LIN {X 0,Y 340.767,Z 675.84,A -85,B 0,C 180,E1 -14245.664,E2 -14245.664} C_VEL
LIN {X 0,Y 340.733,Z 675.796,A -85,B 0,C 180,E1 -14248.32,E2 -14248.32} C_VEL
LIN {X 0,Y 340.696,Z 675.835,A -85,B 0,C 180,E1 -14251.044,E2 -14251.044} C_VEL
LIN {X 0,Y 340.71,Z 675.812,A -85,B 0,C 180,E1 -14255.279,E2 -14255.279} C_VEL
LIN {X 0,Y 340.71,Z 675.84,A -85,B 0,C 180,E1 -14258.388,E2 -14258.388} C_VEL
LIN {X 0,Y 340.718,Z 675.858,A -85,B 0,C 180,E1 -14261.304,E2 -14261.304} C_VEL
LIN {X 0,Y 340.716,Z 675.858,A -85,B 0,C 180,E1 -14264.532,E2 -14264.532} C_VEL
LIN {X 0,Y 340.727,Z 675.857,A -85,B 0,C 180,E1 -14267.949,E2 -14267.949} C_VEL
LIN {X 0,Y 340.758,Z 676.06,A -85,B 0,C 180,E1 -14271.835,E2 -14271.835} C_VEL
LIN {X 0,Y 341.027,Z 677.234,A -85,B 0,C 180,E1 -14272.318,E2 -14272.318} C_VEL
LIN {X 0,Y 342.41,Z 679.667,A -85,B 0,C 180,E1 -14272.976,E2 -14272.976} C_VEL
LIN {X 0,Y 344.684,Z 681.388,A -85,B 0,C 180,E1 -14273.895,E2 -14273.895} C_VEL
LIN {X 0,Y 345.815,Z 682.281,A -85,B 0,C 180,E1 -14274.381,E2 -14274.381} C_VEL
LIN {X 0,Y 347.437,Z 685.007,A -85,B 0,C 180,E1 -14275.129,E2 -14275.129} C_VEL
LIN {X 0,Y 350.033,Z 687.231,A -85,B 0,C 180,E1 -14276.266,E2 -14276.266} C_VEL
LIN {X 0,Y 351.154,Z 688.02,A -85,B 0,C 180,E1 -14276.744,E2 -14276.744} C_VEL
LIN {X 0,Y 353.08,Z 690.98,A -85,B 0,C 180,E1 -14277.691,E2 -14277.691} C_VEL
LIN {X 0,Y 355.654,Z 693.147,A -85,B 0,C 180,E1 -14278.882,E2 -14278.882} C_VEL
LIN {X 0,Y 357.002,Z 694.101,A -85,B 0,C 180,E1 -14279.493,E2 -14279.493} C_VEL
LIN {X 0,Y 359.425,Z 697.413,A -85,B 0,C 180,E1 -14280.737,E2 -14280.737} C_VEL
LIN {X 0,Y 362.273,Z 699.528,A -85,B 0,C 180,E1 -14282.149,E2 -14282.149} C_VEL
LIN {X 0,Y 363.124,Z 700.378,A -85,B 0,C 180,E1 -14282.611,E2 -14282.611} C_VEL
LIN {X 0,Y 365.113,Z 703.18,A -85,B 0,C 180,E1 -14283.723,E2 -14283.723} C_VEL
LIN {X 0,Y 367.846,Z 705.386,A -85,B 0,C 180,E1 -14285.232,E2 -14285.232} C_VEL
LIN {X 0,Y 369.089,Z 706.243,A -85,B 0,C 180,E1 -14285.932,E2 -14285.932} C_VEL
LIN {X 0,Y 371.469,Z 709.532,A -85,B 0,C 180,E1 -14287.437,E2 -14287.437} C_VEL
LIN {X 0,Y 374.201,Z 711.633,A -85,B 0,C 180,E1 -14289.17,E2 -14289.17} C_VEL
LIN {X 0,Y 375.879,Z 712.69,A -85,B 0,C 180,E1 -14290.269,E2 -14290.269} C_VEL
LIN {X 0,Y 377.819,Z 715.534,A -85,B 0,C 180,E1 -14291.772,E2 -14291.772} C_VEL
LIN {X 0,Y 380.32,Z 717.676,A -85,B 0,C 180,E1 -14293.763,E2 -14293.763} C_VEL
LIN {X 0,Y 382.812,Z 719.086,A -85,B 0,C 180,E1 -14295.905,E2 -14295.905} C_VEL
LIN {X 0,Y 384.247,Z 721.472,A -85,B 0,C 180,E1 -14297.505,E2 -14297.505} C_VEL
LIN {X 0,Y 386.099,Z 723.313,A -85,B 0,C 180,E1 -14299.68,E2 -14299.68} C_VEL
LIN {X 0,Y 387.892,Z 724.36,A -85,B 0,C 180,E1 -14302.256,E2 -14302.256} C_VEL
LIN {X 0,Y 389.273,Z 725.077,A -85,B 0,C 180,E1 -14305.045,E2 -14305.045} C_VEL
LIN {X 0,Y 390.059,Z 725.483,A -85,B 0,C 180,E1 -14307.935,E2 -14307.935} C_VEL
LIN {X 0,Y 390.26,Z 725.548,A -85,B 0,C 180,E1 -14310,E2 -14310} C_VEL
LIN {X 0,Y 390.059,Z 725.486,A -85,B 0,C 180,E1 -14312.065,E2 -14312.065} C_VEL
LIN {X 0,Y 389.272,Z 725.078,A -85,B 0,C 180,E1 -14314.953,E2 -14314.953} C_VEL
LIN {X 0,Y 387.893,Z 724.36,A -85,B 0,C 180,E1 -14317.744,E2 -14317.744} C_VEL
LIN {X 0,Y 386.1,Z 723.319,A -85,B 0,C 180,E1 -14320.32,E2 -14320.32} C_VEL
LIN {X 0,Y 384.178,Z 721.341,A -85,B 0,C 180,E1 -14322.58,E2 -14322.58} C_VEL
LIN {X 0,Y 382.562,Z 718.807,A -85,B 0,C 180,E1 -14324.348,E2 -14324.348} C_VEL
LIN {X 0,Y 379.559,Z 717.133,A -85,B 0,C 180,E1 -14326.866,E2 -14326.866} C_VEL
LIN {X 0,Y 377.187,Z 714.751,A -85,B 0,C 180,E1 -14328.707,E2 -14328.707} C_VEL
LIN {X 0,Y 375.566,Z 712.349,A -85,B 0,C 180,E1 -14329.944,E2 -14329.944} C_VEL
LIN {X 0,Y 372.385,Z 710.399,A -85,B 0,C 180,E1 -14331.974,E2 -14331.974} C_VEL
LIN {X 0,Y 369.885,Z 707.552,A -85,B 0,C 180,E1 -14333.563,E2 -14333.563} C_VEL
LIN {X 0,Y 368.864,Z 705.955,A -85,B 0,C 180,E1 -14334.201,E2 -14334.201} C_VEL
LIN {X 0,Y 365.884,Z 703.986,A -85,B 0,C 180,E1 -14335.838,E2 -14335.838} C_VEL
LIN {X 0,Y 363.626,Z 701.259,A -85,B 0,C 180,E1 -14337.098,E2 -14337.098} C_VEL
LIN {X 0,Y 362.729,Z 699.764,A -85,B 0,C 180,E1 -14337.62,E2 -14337.62} C_VEL
LIN {X 0,Y 359.826,Z 697.815,A -85,B 0,C 180,E1 -14339.06,E2 -14339.06} C_VEL
LIN {X 0,Y 357.355,Z 694.737,A -85,B 0,C 180,E1 -14340.312,E2 -14340.312} C_VEL
LIN {X 0,Y 356.555,Z 693.62,A -85,B 0,C 180,E1 -14340.722,E2 -14340.722} C_VEL
LIN {X 0,Y 353.621,Z 691.552,A -85,B 0,C 180,E1 -14342.065,E2 -14342.065} C_VEL
LIN {X 0,Y 351.546,Z 688.772,A -85,B 0,C 180,E1 -14343.05,E2 -14343.05} C_VEL
LIN {X 0,Y 350.95,Z 687.687,A -85,B 0,C 180,E1 -14343.357,E2 -14343.357} C_VEL
LIN {X 0,Y 347.992,Z 685.635,A -85,B 0,C 180,E1 -14344.624,E2 -14344.624} C_VEL
LIN {X 0,Y 346.203,Z 683.113,A -85,B 0,C 180,E1 -14345.429,E2 -14345.429} C_VEL
LIN {X 0,Y 345.49,Z 681.814,A -85,B 0,C 180,E1 -14345.769,E2 -14345.769} C_VEL
LIN {X 0,Y 342.717,Z 679.998,A -85,B 0,C 180,E1 -14346.894,E2 -14346.894} C_VEL
LIN {X 0,Y 341.161,Z 677.596,A -85,B 0,C 180,E1 -14347.61,E2 -14347.61} C_VEL
LIN {X 0,Y 340.803,Z 676.233,A -85,B 0,C 180,E1 -14348.043,E2 -14348.043} C_VEL
LIN {X 0,Y 340.72,Z 675.904,A -85,B 0,C 180,E1 -14348.389,E2 -14348.389} C_VEL
LIN {X 0,Y 340.727,Z 675.857,A -85,B 0,C 180,E1 -14352.051,E2 -14352.051} C_VEL
LIN {X 0,Y 340.716,Z 675.858,A -85,B 0,C 180,E1 -14355.468,E2 -14355.468} C_VEL
LIN {X 0,Y 340.718,Z 675.858,A -85,B 0,C 180,E1 -14358.696,E2 -14358.696} C_VEL
LIN {X 0,Y 340.731,Z 675.833,A -85,B 0,C 180,E1 -14361.773,E2 -14361.773} C_VEL
LIN {X 0,Y 340.715,Z 675.827,A -85,B 0,C 180,E1 -14365.595,E2 -14365.595} C_VEL
LIN {X 0,Y 340.715,Z 675.816,A -85,B 0,C 180,E1 -14369.568,E2 -14369.568} C_VEL
LIN {X 0,Y 340.797,Z 675.806,A -85,B 0,C 180,E1 -14373.02,E2 -14373.02} C_VEL
LIN {X 0,Y 340.757,Z 675.844,A -85,B 0,C 180,E1 -14374.692,E2 -14374.692} C_VEL
LIN {X 0,Y 340.082,Z 675.936,A -85,B 0,C 180,E1 -14375.679,E2 -14375.679} C_VEL
LIN {X 0,Y 337.203,Z 676.292,A -85,B 0,C 180,E1 -14377.284,E2 -14377.284} C_VEL
LIN {X 0,Y 334.787,Z 676.588,A -85,B 0,C 180,E1 -14378.584,E2 -14378.584} C_VEL
LIN {X 0,Y 333.782,Z 676.719,A -85,B 0,C 180,E1 -14379.591,E2 -14379.591} C_VEL
LIN {X 0,Y 333.717,Z 676.723,A -85,B 0,C 180,E1 -14379.931,E2 -14379.931} C_VEL
LIN {X 0,Y 333.737,Z 676.708,A -85,B 0,C 180,E1 -14382.854,E2 -14382.854} C_VEL
LIN {X 0,Y 333.788,Z 676.698,A -85,B 0,C 180,E1 -14386.609,E2 -14386.609} C_VEL
LIN {X 0,Y 333.853,Z 676.706,A -85,B 0,C 180,E1 -14390.305,E2 -14390.305} C_VEL
LIN {X 0,Y 334.006,Z 676.673,A -85,B 0,C 180,E1 -14392.747,E2 -14392.747} C_VEL
LIN {X 0,Y 333.807,Z 676.714,A -85,B 0,C 180,E1 -14395.169,E2 -14395.169} C_VEL
LIN {X 0,Y 334.099,Z 676.658,A -85,B 0,C 180,E1 -14397.589,E2 -14397.589} C_VEL
LIN {X 0,Y 334.259,Z 676.66,A -85,B 0,C 180,E1 -14400,E2 -14400} C_VEL
LIN {X 0,Y 334.099,Z 676.662,A -85,B 0,C 180,E1 -14402.412,E2 -14402.412} C_VEL
LIN {X 0,Y 334.012,Z 676.688,A -85,B 0,C 180,E1 -14406.039,E2 -14406.039} C_VEL
LIN {X 0,Y 333.977,Z 676.673,A -85,B 0,C 180,E1 -14408.502,E2 -14408.502} C_VEL
LIN {X 0,Y 333.788,Z 676.703,A -85,B 0,C 180,E1 -14412.155,E2 -14412.155} C_VEL
LIN {X 0,Y 333.77,Z 676.718,A -85,B 0,C 180,E1 -14415.887,E2 -14415.887} C_VEL
LIN {X 0,Y 333.79,Z 676.705,A -85,B 0,C 180,E1 -14418.656,E2 -14418.656} C_VEL
LIN {X 0,Y 333.686,Z 676.715,A -85,B 0,C 180,E1 -14422.279,E2 -14422.279} C_VEL
LIN {X 0,Y 333.729,Z 676.704,A -85,B 0,C 180,E1 -14426.247,E2 -14426.247} C_VEL
LIN {X 0,Y 333.705,Z 676.667,A -85,B 0,C 180,E1 -14428.973,E2 -14428.973} C_VEL
LIN {X 0,Y 333.637,Z 676.739,A -85,B 0,C 180,E1 -14432.588,E2 -14432.588} C_VEL
LIN {X 0,Y 333.672,Z 676.695,A -85,B 0,C 180,E1 -14436.14,E2 -14436.14} C_VEL
LIN {X 0,Y 333.68,Z 676.726,A -85,B 0,C 180,E1 -14439.188,E2 -14439.188} C_VEL
LIN {X 0,Y 333.735,Z 676.913,A -85,B 0,C 180,E1 -14443.009,E2 -14443.009} C_VEL
LIN {X 0,Y 336.743,Z 686.921,A -85,B 0,C 180,E1 -14446.472,E2 -14446.472} C_VEL
LIN {X 0,Y 337.307,Z 688.603,A -85,B 0,C 180,E1 -14446.878,E2 -14446.878} C_VEL
LIN {X 0,Y 339.979,Z 693.107,A -85,B 0,C 180,E1 -14447.437,E2 -14447.437} C_VEL
LIN {X 0,Y 348.642,Z 708.555,A -85,B 0,C 180,E1 -14449.135,E2 -14449.135} C_VEL
LIN {X 0,Y 357.092,Z 725,A -85,B 0,C 180,E1 -14450.708,E2 -14450.708} C_VEL
LIN {X 0,Y 363.501,Z 738.717,A -85,B 0,C 180,E1 -14451.861,E2 -14451.861} C_VEL
LIN {X 0,Y 365.531,Z 748.623,A -85,B 0,C 180,E1 -14452.349,E2 -14452.349} C_VEL
LIN {X 0,Y 360.507,Z 891.622,A -85,B 0,C 180,E1 -14455.234,E2 -14455.234} C_VEL
LIN {X 0,Y 359.774,Z 902.847,A -85,B 0,C 180,E1 -14455.537,E2 -14455.537} C_VEL
LIN {X 0,Y 358.362,Z 917.16,A -85,B 0,C 180,E1 -14456.062,E2 -14456.062} C_VEL
LIN {X 0,Y 356.831,Z 930.278,A -85,B 0,C 180,E1 -14456.702,E2 -14456.702} C_VEL
LIN {X 0,Y 355.352,Z 941.666,A -85,B 0,C 180,E1 -14457.39,E2 -14457.39} C_VEL
LIN {X 0,Y 353.249,Z 954.9,A -85,B 0,C 180,E1 -14458.35,E2 -14458.35} C_VEL
LIN {X 0,Y 351.239,Z 966.54,A -85,B 0,C 180,E1 -14459.361,E2 -14459.361} C_VEL
LIN {X 0,Y 348.937,Z 978.635,A -85,B 0,C 180,E1 -14460.598,E2 -14460.598} C_VEL
LIN {X 0,Y 346.666,Z 989.433,A -85,B 0,C 180,E1 -14461.879,E2 -14461.879} C_VEL
LIN {X 0,Y 344.484,Z 999.934,A -85,B 0,C 180,E1 -14463.332,E2 -14463.332} C_VEL
LIN {X 0,Y 342.425,Z 1009.204,A -85,B 0,C 180,E1 -14464.795,E2 -14464.795} C_VEL
LIN {X 0,Y 340.254,Z 1018.938,A -85,B 0,C 180,E1 -14466.572,E2 -14466.572} C_VEL
LIN {X 0,Y 338.341,Z 1027.463,A -85,B 0,C 180,E1 -14468.365,E2 -14468.365} C_VEL
LIN {X 0,Y 336.521,Z 1036.066,A -85,B 0,C 180,E1 -14470.48,E2 -14470.48} C_VEL
LIN {X 0,Y 335.246,Z 1042.499,A -85,B 0,C 180,E1 -14472.304,E2 -14472.304} C_VEL
LIN {X 0,Y 333.919,Z 1049.762,A -85,B 0,C 180,E1 -14474.747,E2 -14474.747} C_VEL
LIN {X 0,Y 333.001,Z 1055.764,A -85,B 0,C 180,E1 -14477.197,E2 -14477.197} C_VEL
LIN {X 0,Y 332.475,Z 1059.512,A -85,B 0,C 180,E1 -14479.033,E2 -14479.033} C_VEL
LIN {X 0,Y 332.12,Z 1063.512,A -85,B 0,C 180,E1 -14481.482,E2 -14481.482} C_VEL
LIN {X 0,Y 332.03,Z 1066.47,A -85,B 0,C 180,E1 -14483.925,E2 -14483.925} C_VEL
LIN {X 0,Y 331.937,Z 1067.654,A -85,B 0,C 180,E1 -14485.142,E2 -14485.142} C_VEL
LIN {X 0,Y 331.902,Z 1069.122,A -85,B 0,C 180,E1 -14487.573,E2 -14487.573} C_VEL
LIN {X 0,Y 331.967,Z 1069.61,A -85,B 0,C 180,E1 -14490,E2 -14490} C_VEL
LIN {X 0,Y 331.902,Z 1069.122,A -85,B 0,C 180,E1 -14492.427,E2 -14492.427} C_VEL
LIN {X 0,Y 331.937,Z 1067.654,A -85,B 0,C 180,E1 -14494.858,E2 -14494.858} C_VEL
LIN {X 0,Y 332.033,Z 1065.187,A -85,B 0,C 180,E1 -14497.296,E2 -14497.296} C_VEL
LIN {X 0,Y 332.366,Z 1060.601,A -85,B 0,C 180,E1 -14500.354,E2 -14500.354} C_VEL
LIN {X 0,Y 332.844,Z 1057.113,A -85,B 0,C 180,E1 -14502.189,E2 -14502.189} C_VEL
LIN {X 0,Y 333.648,Z 1051.384,A -85,B 0,C 180,E1 -14504.641,E2 -14504.641} C_VEL
LIN {X 0,Y 334.492,Z 1046.322,A -85,B 0,C 180,E1 -14506.478,E2 -14506.478} C_VEL
LIN {X 0,Y 336.142,Z 1038.291,A -85,B 0,C 180,E1 -14508.909,E2 -14508.909} C_VEL
LIN {X 0,Y 337.514,Z 1031.303,A -85,B 0,C 180,E1 -14510.731,E2 -14510.731} C_VEL
LIN {X 0,Y 339.275,Z 1023.335,A -85,B 0,C 180,E1 -14512.533,E2 -14512.533} C_VEL
LIN {X 0,Y 341.369,Z 1014.223,A -85,B 0,C 180,E1 -14514.314,E2 -14514.314} C_VEL
LIN {X 0,Y 343.379,Z 1004.797,A -85,B 0,C 180,E1 -14515.926,E2 -14515.926} C_VEL
LIN {X 0,Y 345.819,Z 993.788,A -85,B 0,C 180,E1 -14517.538,E2 -14517.538} C_VEL
LIN {X 0,Y 347.827,Z 983.618,A -85,B 0,C 180,E1 -14518.842,E2 -14518.842} C_VEL
LIN {X 0,Y 350.215,Z 971.952,A -85,B 0,C 180,E1 -14520.111,E2 -14520.111} C_VEL
LIN {X 0,Y 352.395,Z 959.927,A -85,B 0,C 180,E1 -14521.233,E2 -14521.233} C_VEL
LIN {X 0,Y 354.42,Z 947.608,A -85,B 0,C 180,E1 -14522.202,E2 -14522.202} C_VEL
LIN {X 0,Y 356.268,Z 935.066,A -85,B 0,C 180,E1 -14523.02,E2 -14523.02} C_VEL
LIN {X 0,Y 357.772,Z 922.382,A -85,B 0,C 180,E1 -14523.705,E2 -14523.705} C_VEL
LIN {X 0,Y 359.234,Z 908.721,A -85,B 0,C 180,E1 -14524.267,E2 -14524.267} C_VEL
LIN {X 0,Y 360.331,Z 895.291,A -85,B 0,C 180,E1 -14524.675,E2 -14524.675} C_VEL
LIN {X 0,Y 361.357,Z 868.673,A -85,B 0,C 180,E1 -14525.251,E2 -14525.251} C_VEL
LIN {X 0,Y 365.514,Z 748.139,A -85,B 0,C 180,E1 -14527.664,E2 -14527.664} C_VEL
LIN {X 0,Y 363.359,Z 738.48,A -85,B 0,C 180,E1 -14528.162,E2 -14528.162} C_VEL
LIN {X 0,Y 356.031,Z 722.733,A -85,B 0,C 180,E1 -14529.489,E2 -14529.489} C_VEL
LIN {X 0,Y 346.856,Z 705.28,A -85,B 0,C 180,E1 -14531.207,E2 -14531.207} C_VEL
LIN {X 0,Y 342.028,Z 696.763,A -85,B 0,C 180,E1 -14532.149,E2 -14532.149} C_VEL
LIN {X 0,Y 338.511,Z 690.985,A -85,B 0,C 180,E1 -14532.85,E2 -14532.85} C_VEL
LIN {X 0,Y 337.023,Z 687.928,A -85,B 0,C 180,E1 -14533.239,E2 -14533.239} C_VEL
LIN {X 0,Y 334.479,Z 679.341,A -85,B 0,C 180,E1 -14536.101,E2 -14536.101} C_VEL
LIN {X 0,Y 333.719,Z 676.748,A -85,B 0,C 180,E1 -14537.114,E2 -14537.114} C_VEL
LIN {X 0,Y 333.68,Z 676.726,A -85,B 0,C 180,E1 -14540.812,E2 -14540.812} C_VEL
LIN {X 0,Y 333.672,Z 676.695,A -85,B 0,C 180,E1 -14543.86,E2 -14543.86} C_VEL
LIN {X 0,Y 333.637,Z 676.739,A -85,B 0,C 180,E1 -14547.412,E2 -14547.412} C_VEL
LIN {X 0,Y 333.705,Z 676.667,A -85,B 0,C 180,E1 -14551.027,E2 -14551.027} C_VEL
LIN {X 0,Y 333.729,Z 676.704,A -85,B 0,C 180,E1 -14553.753,E2 -14553.753} C_VEL
LIN {X 0,Y 333.713,Z 676.712,A -85,B 0,C 180,E1 -14557.913,E2 -14557.913} C_VEL
LIN {X 0,Y 333.787,Z 676.704,A -85,B 0,C 180,E1 -14561.589,E2 -14561.589} C_VEL
LIN {X 0,Y 333.801,Z 676.712,A -85,B 0,C 180,E1 -14565.576,E2 -14565.576} C_VEL
LIN {X 0,Y 333.83,Z 676.712,A -85,B 0,C 180,E1 -14569.078,E2 -14569.078} C_VEL
LIN {X 0,Y 334.008,Z 676.671,A -85,B 0,C 180,E1 -14572.747,E2 -14572.747} C_VEL
LIN {X 0,Y 333.807,Z 676.713,A -85,B 0,C 180,E1 -14575.169,E2 -14575.169} C_VEL
LIN {X 0,Y 334.099,Z 676.66,A -85,B 0,C 180,E1 -14577.588,E2 -14577.588} C_VEL
LIN {X 0,Y 334.259,Z 676.659,A -85,B 0,C 180,E1 -14580,E2 -14580} C_VEL
LIN {X 0,Y 334.099,Z 676.658,A -85,B 0,C 180,E1 -14582.411,E2 -14582.411} C_VEL
LIN {X 0,Y 333.99,Z 676.681,A -85,B 0,C 180,E1 -14586.597,E2 -14586.597} C_VEL
LIN {X 0,Y 333.853,Z 676.708,A -85,B 0,C 180,E1 -14589.695,E2 -14589.695} C_VEL
LIN {X 0,Y 333.788,Z 676.699,A -85,B 0,C 180,E1 -14593.391,E2 -14593.391} C_VEL
LIN {X 0,Y 333.737,Z 676.709,A -85,B 0,C 180,E1 -14597.146,E2 -14597.146} C_VEL
LIN {X 0,Y 333.745,Z 676.723,A -85,B 0,C 180,E1 -14599.689,E2 -14599.689} C_VEL
LIN {X 0,Y 333.682,Z 676.727,A -85,B 0,C 180,E1 -14603.589,E2 -14603.589} C_VEL
LIN {X 0,Y 333.729,Z 676.704,A -85,B 0,C 180,E1 -14606.246,E2 -14606.246} C_VEL
LIN {X 0,Y 333.703,Z 676.669,A -85,B 0,C 180,E1 -14608.972,E2 -14608.972} C_VEL
LIN {X 0,Y 333.635,Z 676.741,A -85,B 0,C 180,E1 -14612.587,E2 -14612.587} C_VEL
LIN {X 0,Y 333.668,Z 676.683,A -85,B 0,C 180,E1 -14616.139,E2 -14616.139} C_VEL
LIN {X 0,Y 333.677,Z 676.734,A -85,B 0,C 180,E1 -14619.187,E2 -14619.187} C_VEL
LIN {X 0,Y 333.682,Z 676.734,A -85,B 0,C 180,E1 -14622.511,E2 -14622.511} C_VEL
LIN {X 0,Y 333.653,Z 676.738,A -85,B 0,C 180,E1 -14625.966,E2 -14625.966} C_VEL
LIN {X 0,Y 333.664,Z 676.864,A -85,B 0,C 180,E1 -14629.311,E2 -14629.311} C_VEL
LIN {X 0,Y 333.971,Z 678.117,A -85,B 0,C 180,E1 -14629.854,E2 -14629.854} C_VEL
LIN {X 0,Y 335.547,Z 680.762,A -85,B 0,C 180,E1 -14630.557,E2 -14630.557} C_VEL
LIN {X 0,Y 337.901,Z 682.418,A -85,B 0,C 180,E1 -14631.471,E2 -14631.471} C_VEL
LIN {X 0,Y 338.694,Z 683.215,A -85,B 0,C 180,E1 -14631.798,E2 -14631.798} C_VEL
LIN {X 0,Y 340.556,Z 686.154,A -85,B 0,C 180,E1 -14632.605,E2 -14632.605} C_VEL
LIN {X 0,Y 343.114,Z 688.192,A -85,B 0,C 180,E1 -14633.656,E2 -14633.656} C_VEL
LIN {X 0,Y 343.878,Z 688.778,A -85,B 0,C 180,E1 -14633.965,E2 -14633.965} C_VEL
LIN {X 0,Y 345.866,Z 691.831,A -85,B 0,C 180,E1 -14634.885,E2 -14634.885} C_VEL
LIN {X 0,Y 348.611,Z 694.083,A -85,B 0,C 180,E1 -14636.069,E2 -14636.069} C_VEL
LIN {X 0,Y 349.514,Z 694.878,A -85,B 0,C 180,E1 -14636.459,E2 -14636.459} C_VEL
LIN {X 0,Y 351.608,Z 697.789,A -85,B 0,C 180,E1 -14637.462,E2 -14637.462} C_VEL
LIN {X 0,Y 354.424,Z 700.091,A -85,B 0,C 180,E1 -14638.749,E2 -14638.749} C_VEL
LIN {X 0,Y 355.498,Z 701.01,A -85,B 0,C 180,E1 -14639.245,E2 -14639.245} C_VEL
LIN {X 0,Y 358.132,Z 704.346,A -85,B 0,C 180,E1 -14640.574,E2 -14640.574} C_VEL
LIN {X 0,Y 361.588,Z 707.043,A -85,B 0,C 180,E1 -14642.286,E2 -14642.286} C_VEL
LIN {X 0,Y 363.832,Z 710.035,A -85,B 0,C 180,E1 -14643.526,E2 -14643.526} C_VEL
LIN {X 0,Y 366.633,Z 712.293,A -85,B 0,C 180,E1 -14645.058,E2 -14645.058} C_VEL
LIN {X 0,Y 367.789,Z 713.203,A -85,B 0,C 180,E1 -14645.724,E2 -14645.724} C_VEL
LIN {X 0,Y 370.207,Z 716.399,A -85,B 0,C 180,E1 -14647.233,E2 -14647.233} C_VEL
LIN {X 0,Y 373.102,Z 718.587,A -85,B 0,C 180,E1 -14649.03,E2 -14649.03} C_VEL
LIN {X 0,Y 374.671,Z 719.597,A -85,B 0,C 180,E1 -14650.072,E2 -14650.072} C_VEL
LIN {X 0,Y 376.704,Z 722.459,A -85,B 0,C 180,E1 -14651.607,E2 -14651.607} C_VEL
LIN {X 0,Y 379.384,Z 724.71,A -85,B 0,C 180,E1 -14653.722,E2 -14653.722} C_VEL
LIN {X 0,Y 381.803,Z 726.129,A -85,B 0,C 180,E1 -14655.785,E2 -14655.785} C_VEL
LIN {X 0,Y 383.338,Z 728.552,A -85,B 0,C 180,E1 -14657.475,E2 -14657.475} C_VEL
LIN {X 0,Y 385.21,Z 730.362,A -85,B 0,C 180,E1 -14659.656,E2 -14659.656} C_VEL
LIN {X 0,Y 387.012,Z 731.404,A -85,B 0,C 180,E1 -14662.239,E2 -14662.239} C_VEL
LIN {X 0,Y 388.405,Z 732.112,A -85,B 0,C 180,E1 -14665.034,E2 -14665.034} C_VEL
LIN {X 0,Y 389.194,Z 732.531,A -85,B 0,C 180,E1 -14667.93,E2 -14667.93} C_VEL
LIN {X 0,Y 389.395,Z 732.596,A -85,B 0,C 180,E1 -14670,E2 -14670} C_VEL
LIN {X 0,Y 389.194,Z 732.534,A -85,B 0,C 180,E1 -14672.07,E2 -14672.07} C_VEL
LIN {X 0,Y 388.402,Z 732.127,A -85,B 0,C 180,E1 -14674.965,E2 -14674.965} C_VEL
LIN {X 0,Y 387.012,Z 731.404,A -85,B 0,C 180,E1 -14677.762,E2 -14677.762} C_VEL
LIN {X 0,Y 385.211,Z 730.37,A -85,B 0,C 180,E1 -14680.344,E2 -14680.344} C_VEL
LIN {X 0,Y 383.262,Z 728.47,A -85,B 0,C 180,E1 -14682.611,E2 -14682.611} C_VEL
LIN {X 0,Y 381.464,Z 725.733,A -85,B 0,C 180,E1 -14684.549,E2 -14684.549} C_VEL
LIN {X 0,Y 378.624,Z 724.167,A -85,B 0,C 180,E1 -14686.909,E2 -14686.909} C_VEL
LIN {X 0,Y 376.102,Z 721.752,A -85,B 0,C 180,E1 -14688.835,E2 -14688.835} C_VEL
LIN {X 0,Y 374.328,Z 719.256,A -85,B 0,C 180,E1 -14690.159,E2 -14690.159} C_VEL
LIN {X 0,Y 371.046,Z 717.139,A -85,B 0,C 180,E1 -14692.26,E2 -14692.26} C_VEL
LIN {X 0,Y 368.347,Z 714.068,A -85,B 0,C 180,E1 -14693.936,E2 -14693.936} C_VEL
LIN {X 0,Y 367.399,Z 712.765,A -85,B 0,C 180,E1 -14694.507,E2 -14694.507} C_VEL
LIN {X 0,Y 364.032,Z 710.284,A -85,B 0,C 180,E1 -14696.361,E2 -14696.361} C_VEL
LIN {X 0,Y 361.497,Z 706.91,A -85,B 0,C 180,E1 -14697.767,E2 -14697.767} C_VEL
LIN {X 0,Y 357.983,Z 704.195,A -85,B 0,C 180,E1 -14699.498,E2 -14699.498} C_VEL
LIN {X 0,Y 355.428,Z 700.878,A -85,B 0,C 180,E1 -14700.791,E2 -14700.791} C_VEL
LIN {X 0,Y 351.604,Z 697.812,A -85,B 0,C 180,E1 -14702.538,E2 -14702.538} C_VEL
LIN {X 0,Y 349.346,Z 694.606,A -85,B 0,C 180,E1 -14703.619,E2 -14703.619} C_VEL
LIN {X 0,Y 345.974,Z 691.939,A -85,B 0,C 180,E1 -14705.069,E2 -14705.069} C_VEL
LIN {X 0,Y 343.987,Z 688.966,A -85,B 0,C 180,E1 -14705.984,E2 -14705.984} C_VEL
LIN {X 0,Y 343.481,Z 688.356,A -85,B 0,C 180,E1 -14706.205,E2 -14706.205} C_VEL
LIN {X 0,Y 340.706,Z 686.315,A -85,B 0,C 180,E1 -14707.33,E2 -14707.33} C_VEL
LIN {X 0,Y 338.768,Z 683.404,A -85,B 0,C 180,E1 -14708.167,E2 -14708.167} C_VEL
LIN {X 0,Y 338.123,Z 682.497,A -85,B 0,C 180,E1 -14708.445,E2 -14708.445} C_VEL
LIN {X 0,Y 335.75,Z 680.971,A -85,B 0,C 180,E1 -14709.364,E2 -14709.364} C_VEL
LIN {X 0,Y 334.088,Z 678.423,A -85,B 0,C 180,E1 -14710.083,E2 -14710.083} C_VEL
LIN {X 0,Y 333.717,Z 677.051,A -85,B 0,C 180,E1 -14710.56,E2 -14710.56} C_VEL
LIN {X 0,Y 333.678,Z 676.81,A -85,B 0,C 180,E1 -14710.761,E2 -14710.761} C_VEL
LIN {X 0,Y 333.656,Z 676.738,A -85,B 0,C 180,E1 -14714.262,E2 -14714.262} C_VEL
LIN {X 0,Y 333.687,Z 676.734,A -85,B 0,C 180,E1 -14717.626,E2 -14717.626} C_VEL
LIN {X 0,Y 333.675,Z 676.727,A -85,B 0,C 180,E1 -14721.195,E2 -14721.195} C_VEL
LIN {X 0,Y 333.677,Z 676.695,A -85,B 0,C 180,E1 -14725.226,E2 -14725.226} C_VEL
LIN {X 0,Y 333.625,Z 676.733,A -85,B 0,C 180,E1 -14728.222,E2 -14728.222} C_VEL
LIN {X 0,Y 333.703,Z 676.67,A -85,B 0,C 180,E1 -14731.028,E2 -14731.028} C_VEL
LIN {X 0,Y 333.709,Z 676.723,A -85,B 0,C 180,E1 -14734.697,E2 -14734.697} C_VEL
LIN {X 0,Y 333.713,Z 676.714,A -85,B 0,C 180,E1 -14737.913,E2 -14737.913} C_VEL
LIN {X 0,Y 333.717,Z 676.723,A -85,B 0,C 180,E1 -14739.931,E2 -14739.931} C_VEL
LIN {X 0,Y 333.094,Z 676.806,A -85,B 0,C 180,E1 -14740.938,E2 -14740.938} C_VEL
LIN {X 0,Y 330.26,Z 677.162,A -85,B 0,C 180,E1 -14742.577,E2 -14742.577} C_VEL
LIN {X 0,Y 327.844,Z 677.461,A -85,B 0,C 180,E1 -14743.905,E2 -14743.905} C_VEL
LIN {X 0,Y 326.823,Z 677.584,A -85,B 0,C 180,E1 -14744.932,E2 -14744.932} C_VEL
LIN {X 0,Y 326.749,Z 677.591,A -85,B 0,C 180,E1 -14745.28,E2 -14745.28} C_VEL
LIN {X 0,Y 326.761,Z 677.587,A -85,B 0,C 180,E1 -14748.839,E2 -14748.839} C_VEL
LIN {X 0,Y 326.959,Z 677.549,A -85,B 0,C 180,E1 -14752.59,E2 -14752.59} C_VEL
LIN {X 0,Y 326.774,Z 677.591,A -85,B 0,C 180,E1 -14755.065,E2 -14755.065} C_VEL
LIN {X 0,Y 327.04,Z 677.537,A -85,B 0,C 180,E1 -14757.537,E2 -14757.537} C_VEL
LIN {X 0,Y 327.209,Z 677.539,A -85,B 0,C 180,E1 -14760,E2 -14760} C_VEL
LIN {X 0,Y 327.04,Z 677.54,A -85,B 0,C 180,E1 -14762.464,E2 -14762.464} C_VEL
LIN {X 0,Y 326.987,Z 677.562,A -85,B 0,C 180,E1 -14766.17,E2 -14766.17} C_VEL
LIN {X 0,Y 326.907,Z 677.554,A -85,B 0,C 180,E1 -14768.656,E2 -14768.656} C_VEL
LIN {X 0,Y 326.73,Z 677.579,A -85,B 0,C 180,E1 -14772.422,E2 -14772.422} C_VEL
LIN {X 0,Y 326.747,Z 677.592,A -85,B 0,C 180,E1 -14774.958,E2 -14774.958} C_VEL
LIN {X 0,Y 326.728,Z 677.586,A -85,B 0,C 180,E1 -14778.84,E2 -14778.84} C_VEL
LIN {X 0,Y 326.614,Z 677.596,A -85,B 0,C 180,E1 -14782.788,E2 -14782.788} C_VEL
LIN {X 0,Y 326.684,Z 677.598,A -85,B 0,C 180,E1 -14785.484,E2 -14785.484} C_VEL
LIN {X 0,Y 326.654,Z 677.548,A -85,B 0,C 180,E1 -14789.66,E2 -14789.66} C_VEL
LIN {X 0,Y 326.601,Z 677.593,A -85,B 0,C 180,E1 -14794.02,E2 -14794.02} C_VEL
LIN {X 0,Y 326.625,Z 677.584,A -85,B 0,C 180,E1 -14797.24,E2 -14797.24} C_VEL
LIN {X 0,Y 326.631,Z 677.585,A -85,B 0,C 180,E1 -14800.203,E2 -14800.203} C_VEL
LIN {X 0,Y 326.654,Z 677.674,A -85,B 0,C 180,E1 -14801.966,E2 -14801.966} C_VEL
LIN {X 0,Y 329.322,Z 686.586,A -85,B 0,C 180,E1 -14805.233,E2 -14805.233} C_VEL
LIN {X 0,Y 329.878,Z 688.178,A -85,B 0,C 180,E1 -14805.652,E2 -14805.652} C_VEL
LIN {X 0,Y 333.9,Z 695.082,A -85,B 0,C 180,E1 -14806.536,E2 -14806.536} C_VEL
LIN {X 0,Y 337.305,Z 700.785,A -85,B 0,C 180,E1 -14807.24,E2 -14807.24} C_VEL
LIN {X 0,Y 344.063,Z 712.862,A -85,B 0,C 180,E1 -14808.593,E2 -14808.593} C_VEL
LIN {X 0,Y 352.128,Z 728.696,A -85,B 0,C 180,E1 -14810.145,E2 -14810.145} C_VEL
LIN {X 0,Y 358.283,Z 742.036,A -85,B 0,C 180,E1 -14811.291,E2 -14811.291} C_VEL
LIN {X 0,Y 359.874,Z 750.573,A -85,B 0,C 180,E1 -14811.705,E2 -14811.705} C_VEL
LIN {X 0,Y 354.657,Z 892.216,A -85,B 0,C 180,E1 -14814.6,E2 -14814.6} C_VEL
LIN {X 0,Y 353.947,Z 902.642,A -85,B 0,C 180,E1 -14814.887,E2 -14814.887} C_VEL
LIN {X 0,Y 352.493,Z 916.955,A -85,B 0,C 180,E1 -14815.417,E2 -14815.417} C_VEL
LIN {X 0,Y 350.899,Z 930.072,A -85,B 0,C 180,E1 -14816.063,E2 -14816.063} C_VEL
LIN {X 0,Y 349.366,Z 941.46,A -85,B 0,C 180,E1 -14816.759,E2 -14816.759} C_VEL
LIN {X 0,Y 347.178,Z 954.693,A -85,B 0,C 180,E1 -14817.731,E2 -14817.731} C_VEL
LIN {X 0,Y 344.923,Z 967.242,A -85,B 0,C 180,E1 -14818.845,E2 -14818.845} C_VEL
LIN {X 0,Y 342.727,Z 978.428,A -85,B 0,C 180,E1 -14820.012,E2 -14820.012} C_VEL
LIN {X 0,Y 340.366,Z 989.226,A -85,B 0,C 180,E1 -14821.311,E2 -14821.311} C_VEL
LIN {X 0,Y 338.075,Z 999.726,A -85,B 0,C 180,E1 -14822.785,E2 -14822.785} C_VEL
LIN {X 0,Y 335.737,Z 1009.804,A -85,B 0,C 180,E1 -14824.417,E2 -14824.417} C_VEL
LIN {X 0,Y 333.636,Z 1018.729,A -85,B 0,C 180,E1 -14826.078,E2 -14826.078} C_VEL
LIN {X 0,Y 331.656,Z 1027.254,A -85,B 0,C 180,E1 -14827.906,E2 -14827.906} C_VEL
LIN {X 0,Y 329.739,Z 1035.857,A -85,B 0,C 180,E1 -14830.061,E2 -14830.061} C_VEL
LIN {X 0,Y 328.415,Z 1042.291,A -85,B 0,C 180,E1 -14831.923,E2 -14831.923} C_VEL
LIN {X 0,Y 326.953,Z 1049.553,A -85,B 0,C 180,E1 -14834.414,E2 -14834.414} C_VEL
LIN {X 0,Y 326.226,Z 1054.207,A -85,B 0,C 180,E1 -14836.292,E2 -14836.292} C_VEL
LIN {X 0,Y 325.451,Z 1059.305,A -85,B 0,C 180,E1 -14838.793,E2 -14838.793} C_VEL
LIN {X 0,Y 325.05,Z 1063.305,A -85,B 0,C 180,E1 -14841.295,E2 -14841.295} C_VEL
LIN {X 0,Y 324.944,Z 1066.264,A -85,B 0,C 180,E1 -14843.792,E2 -14843.792} C_VEL
LIN {X 0,Y 324.851,Z 1067.449,A -85,B 0,C 180,E1 -14845.036,E2 -14845.036} C_VEL
LIN {X 0,Y 324.821,Z 1068.917,A -85,B 0,C 180,E1 -14847.52,E2 -14847.52} C_VEL
LIN {X 0,Y 324.871,Z 1069.405,A -85,B 0,C 180,E1 -14850,E2 -14850} C_VEL
LIN {X 0,Y 324.821,Z 1068.917,A -85,B 0,C 180,E1 -14852.48,E2 -14852.48} C_VEL
LIN {X 0,Y 324.851,Z 1067.449,A -85,B 0,C 180,E1 -14854.964,E2 -14854.964} C_VEL
LIN {X 0,Y 324.949,Z 1064.98,A -85,B 0,C 180,E1 -14857.456,E2 -14857.456} C_VEL
LIN {X 0,Y 325.304,Z 1060.393,A -85,B 0,C 180,E1 -14860.581,E2 -14860.581} C_VEL
LIN {X 0,Y 325.805,Z 1056.905,A -85,B 0,C 180,E1 -14862.457,E2 -14862.457} C_VEL
LIN {X 0,Y 326.685,Z 1051.176,A -85,B 0,C 180,E1 -14864.96,E2 -14864.96} C_VEL
LIN {X 0,Y 327.601,Z 1046.113,A -85,B 0,C 180,E1 -14866.834,E2 -14866.834} C_VEL
LIN {X 0,Y 329.318,Z 1038.082,A -85,B 0,C 180,E1 -14869.316,E2 -14869.316} C_VEL
LIN {X 0,Y 330.769,Z 1031.094,A -85,B 0,C 180,E1 -14871.174,E2 -14871.174} C_VEL
LIN {X 0,Y 332.647,Z 1023.127,A -85,B 0,C 180,E1 -14873.007,E2 -14873.007} C_VEL
LIN {X 0,Y 334.826,Z 1014.015,A -85,B 0,C 180,E1 -14874.821,E2 -14874.821} C_VEL
LIN {X 0,Y 336.932,Z 1004.589,A -85,B 0,C 180,E1 -14876.46,E2 -14876.46} C_VEL
LIN {X 0,Y 339.462,Z 993.58,A -85,B 0,C 180,E1 -14878.098,E2 -14878.098} C_VEL
LIN {X 0,Y 341.555,Z 983.411,A -85,B 0,C 180,E1 -14879.423,E2 -14879.423} C_VEL
LIN {X 0,Y 344.042,Z 971.745,A -85,B 0,C 180,E1 -14880.709,E2 -14880.709} C_VEL
LIN {X 0,Y 346.303,Z 959.72,A -85,B 0,C 180,E1 -14881.846,E2 -14881.846} C_VEL
LIN {X 0,Y 348.415,Z 947.402,A -85,B 0,C 180,E1 -14882.826,E2 -14882.826} C_VEL
LIN {X 0,Y 350.308,Z 934.859,A -85,B 0,C 180,E1 -14883.656,E2 -14883.656} C_VEL
LIN {X 0,Y 351.934,Z 921.429,A -85,B 0,C 180,E1 -14884.385,E2 -14884.385} C_VEL
LIN {X 0,Y 353.377,Z 908.515,A -85,B 0,C 180,E1 -14884.917,E2 -14884.917} C_VEL
LIN {X 0,Y 354.543,Z 894.746,A -85,B 0,C 180,E1 -14885.335,E2 -14885.335} C_VEL
LIN {X 0,Y 355.594,Z 868.041,A -85,B 0,C 180,E1 -14885.921,E2 -14885.921} C_VEL
LIN {X 0,Y 359.837,Z 750.412,A -85,B 0,C 180,E1 -14888.304,E2 -14888.304} C_VEL
LIN {X 0,Y 359.168,Z 746.234,A -85,B 0,C 180,E1 -14888.492,E2 -14888.492} C_VEL
LIN {X 0,Y 357.99,Z 741.374,A -85,B 0,C 180,E1 -14888.763,E2 -14888.763} C_VEL
LIN {X 0,Y 351.14,Z 726.549,A -85,B 0,C 180,E1 -14890.045,E2 -14890.045} C_VEL
LIN {X 0,Y 340.924,Z 707.003,A -85,B 0,C 180,E1 -14892.032,E2 -14892.032} C_VEL
LIN {X 0,Y 334.808,Z 696.586,A -85,B 0,C 180,E1 -14893.275,E2 -14893.275} C_VEL
LIN {X 0,Y 331.603,Z 691.28,A -85,B 0,C 180,E1 -14893.95,E2 -14893.95} C_VEL
LIN {X 0,Y 329.633,Z 687.593,A -85,B 0,C 180,E1 -14894.461,E2 -14894.461} C_VEL
LIN {X 0,Y 327.292,Z 679.712,A -85,B 0,C 180,E1 -14897.205,E2 -14897.205} C_VEL
LIN {X 0,Y 326.653,Z 677.641,A -85,B 0,C 180,E1 -14898.067,E2 -14898.067} C_VEL
LIN {X 0,Y 326.643,Z 677.612,A -85,B 0,C 180,E1 -14901.394,E2 -14901.394} C_VEL
LIN {X 0,Y 326.614,Z 677.575,A -85,B 0,C 180,E1 -14904.851,E2 -14904.851} C_VEL
LIN {X 0,Y 326.602,Z 677.616,A -85,B 0,C 180,E1 -14907.455,E2 -14907.455} C_VEL
LIN {X 0,Y 326.654,Z 677.548,A -85,B 0,C 180,E1 -14910.34,E2 -14910.34} C_VEL
LIN {X 0,Y 326.684,Z 677.598,A -85,B 0,C 180,E1 -14914.516,E2 -14914.516} C_VEL
LIN {X 0,Y 326.646,Z 677.597,A -85,B 0,C 180,E1 -14918.545,E2 -14918.545} C_VEL
LIN {X 0,Y 326.738,Z 677.585,A -85,B 0,C 180,E1 -14921.177,E2 -14921.177} C_VEL
LIN {X 0,Y 326.756,Z 677.59,A -85,B 0,C 180,E1 -14925.433,E2 -14925.433} C_VEL
LIN {X 0,Y 326.766,Z 677.589,A -85,B 0,C 180,E1 -14928.839,E2 -14928.839} C_VEL
LIN {X 0,Y 326.961,Z 677.547,A -85,B 0,C 180,E1 -14932.59,E2 -14932.59} C_VEL
LIN {X 0,Y 326.774,Z 677.59,A -85,B 0,C 180,E1 -14935.065,E2 -14935.065} C_VEL
LIN {X 0,Y 327.04,Z 677.539,A -85,B 0,C 180,E1 -14937.536,E2 -14937.536} C_VEL
LIN {X 0,Y 327.209,Z 677.537,A -85,B 0,C 180,E1 -14940,E2 -14940} C_VEL
LIN {X 0,Y 327.04,Z 677.537,A -85,B 0,C 180,E1 -14942.463,E2 -14942.463} C_VEL
LIN {X 0,Y 326.959,Z 677.557,A -85,B 0,C 180,E1 -14946.588,E2 -14946.588} C_VEL
LIN {X 0,Y 326.906,Z 677.562,A -85,B 0,C 180,E1 -14948.655,E2 -14948.655} C_VEL
LIN {X 0,Y 326.725,Z 677.578,A -85,B 0,C 180,E1 -14952.421,E2 -14952.421} C_VEL
LIN {X 0,Y 326.746,Z 677.594,A -85,B 0,C 180,E1 -14954.957,E2 -14954.957} C_VEL
LIN {X 0,Y 326.729,Z 677.588,A -85,B 0,C 180,E1 -14958.84,E2 -14958.84} C_VEL
LIN {X 0,Y 326.619,Z 677.597,A -85,B 0,C 180,E1 -14962.787,E2 -14962.787} C_VEL
LIN {X 0,Y 326.684,Z 677.597,A -85,B 0,C 180,E1 -14965.484,E2 -14965.484} C_VEL
LIN {X 0,Y 326.653,Z 677.551,A -85,B 0,C 180,E1 -14969.659,E2 -14969.659} C_VEL
LIN {X 0,Y 326.599,Z 677.591,A -85,B 0,C 180,E1 -14974.02,E2 -14974.02} C_VEL
LIN {X 0,Y 326.622,Z 677.567,A -85,B 0,C 180,E1 -14977.239,E2 -14977.239} C_VEL
LIN {X 0,Y 326.628,Z 677.613,A -85,B 0,C 180,E1 -14980.203,E2 -14980.203} C_VEL
LIN {X 0,Y 326.613,Z 677.615,A -85,B 0,C 180,E1 -14983.516,E2 -14983.516} C_VEL
LIN {X 0,Y 326.643,Z 677.819,A -85,B 0,C 180,E1 -14987.015,E2 -14987.015} C_VEL
LIN {X 0,Y 326.921,Z 678.872,A -85,B 0,C 180,E1 -14987.478,E2 -14987.478} C_VEL
LIN {X 0,Y 328.385,Z 681.521,A -85,B 0,C 180,E1 -14988.11,E2 -14988.11} C_VEL
LIN {X 0,Y 331.492,Z 683.889,A -85,B 0,C 180,E1 -14989.29,E2 -14989.29} C_VEL
LIN {X 0,Y 333.333,Z 686.892,A -85,B 0,C 180,E1 -14990.071,E2 -14990.071} C_VEL
LIN {X 0,Y 335.93,Z 689.027,A -85,B 0,C 180,E1 -14991.077,E2 -14991.077} C_VEL
LIN {X 0,Y 336.62,Z 689.56,A -85,B 0,C 180,E1 -14991.355,E2 -14991.355} C_VEL
LIN {X 0,Y 338.784,Z 692.779,A -85,B 0,C 180,E1 -14992.291,E2 -14992.291} C_VEL
LIN {X 0,Y 342.122,Z 695.621,A -85,B 0,C 180,E1 -14993.66,E2 -14993.66} C_VEL
LIN {X 0,Y 344.588,Z 698.92,A -85,B 0,C 180,E1 -14994.761,E2 -14994.761} C_VEL
LIN {X 0,Y 347.749,Z 701.507,A -85,B 0,C 180,E1 -14996.118,E2 -14996.118} C_VEL
LIN {X 0,Y 350.248,Z 704.742,A -85,B 0,C 180,E1 -14997.283,E2 -14997.283} C_VEL
LIN {X 0,Y 353.218,Z 707.045,A -85,B 0,C 180,E1 -14998.625,E2 -14998.625} C_VEL
LIN {X 0,Y 354.861,Z 709.053,A -85,B 0,C 180,E1 -14999.418,E2 -14999.418} C_VEL
LIN {X 0,Y 357.946,Z 712.214,A -85,B 0,C 180,E1 -15000.938,E2 -15000.938} C_VEL
LIN {X 0,Y 360.05,Z 713.777,A -85,B 0,C 180,E1 -15001.987,E2 -15001.987} C_VEL
LIN {X 0,Y 362.722,Z 717.132,A -85,B 0,C 180,E1 -15003.438,E2 -15003.438} C_VEL
LIN {X 0,Y 365.766,Z 719.401,A -85,B 0,C 180,E1 -15005.081,E2 -15005.081} C_VEL
LIN {X 0,Y 366.934,Z 720.741,A -85,B 0,C 180,E1 -15005.781,E2 -15005.781} C_VEL
LIN {X 0,Y 369.539,Z 723.799,A -85,B 0,C 180,E1 -15007.381,E2 -15007.381} C_VEL
LIN {X 0,Y 372.776,Z 725.988,A -85,B 0,C 180,E1 -15009.414,E2 -15009.414} C_VEL
LIN {X 0,Y 373.656,Z 726.855,A -85,B 0,C 180,E1 -15010.016,E2 -15010.016} C_VEL
LIN {X 0,Y 375.989,Z 729.746,A -85,B 0,C 180,E1 -15011.739,E2 -15011.739} C_VEL
LIN {X 0,Y 378.644,Z 731.854,A -85,B 0,C 180,E1 -15013.835,E2 -15013.835} C_VEL
LIN {X 0,Y 380.71,Z 733.015,A -85,B 0,C 180,E1 -15015.58,E2 -15015.58} C_VEL
LIN {X 0,Y 382.429,Z 735.625,A -85,B 0,C 180,E1 -15017.445,E2 -15017.445} C_VEL
LIN {X 0,Y 384.306,Z 737.402,A -85,B 0,C 180,E1 -15019.619,E2 -15019.619} C_VEL
LIN {X 0,Y 386.131,Z 738.447,A -85,B 0,C 180,E1 -15022.221,E2 -15022.221} C_VEL
LIN {X 0,Y 387.535,Z 739.162,A -85,B 0,C 180,E1 -15025.023,E2 -15025.023} C_VEL
LIN {X 0,Y 388.329,Z 739.578,A -85,B 0,C 180,E1 -15027.926,E2 -15027.926} C_VEL
LIN {X 0,Y 388.53,Z 739.644,A -85,B 0,C 180,E1 -15030,E2 -15030} C_VEL
LIN {X 0,Y 388.329,Z 739.581,A -85,B 0,C 180,E1 -15032.074,E2 -15032.074} C_VEL
LIN {X 0,Y 387.532,Z 739.176,A -85,B 0,C 180,E1 -15034.976,E2 -15034.976} C_VEL
LIN {X 0,Y 386.131,Z 738.447,A -85,B 0,C 180,E1 -15037.78,E2 -15037.78} C_VEL
LIN {X 0,Y 384.318,Z 737.417,A -85,B 0,C 180,E1 -15040.368,E2 -15040.368} C_VEL
LIN {X 0,Y 382.262,Z 735.441,A -85,B 0,C 180,E1 -15042.745,E2 -15042.745} C_VEL
LIN {X 0,Y 380.379,Z 732.694,A -85,B 0,C 180,E1 -15044.717,E2 -15044.717} C_VEL
LIN {X 0,Y 377.474,Z 731.058,A -85,B 0,C 180,E1 -15047.108,E2 -15047.108} C_VEL
LIN {X 0,Y 374.926,Z 728.605,A -85,B 0,C 180,E1 -15049.036,E2 -15049.036} C_VEL
LIN {X 0,Y 372.992,Z 726.101,A -85,B 0,C 180,E1 -15050.445,E2 -15050.445} C_VEL
LIN {X 0,Y 369.547,Z 723.787,A -85,B 0,C 180,E1 -15052.616,E2 -15052.616} C_VEL
LIN {X 0,Y 366.818,Z 720.628,A -85,B 0,C 180,E1 -15054.286,E2 -15054.286} C_VEL
LIN {X 0,Y 365.94,Z 719.529,A -85,B 0,C 180,E1 -15054.819,E2 -15054.819} C_VEL
LIN {X 0,Y 362.698,Z 717.11,A -85,B 0,C 180,E1 -15056.575,E2 -15056.575} C_VEL
LIN {X 0,Y 360.051,Z 713.787,A -85,B 0,C 180,E1 -15058.013,E2 -15058.013} C_VEL
LIN {X 0,Y 356.268,Z 710.711,A -85,B 0,C 180,E1 -15059.871,E2 -15059.871} C_VEL
LIN {X 0,Y 353.49,Z 707.202,A -85,B 0,C 180,E1 -15061.251,E2 -15061.251} C_VEL
LIN {X 0,Y 350.246,Z 704.754,A -85,B 0,C 180,E1 -15062.717,E2 -15062.717} C_VEL
LIN {X 0,Y 347.673,Z 701.399,A -85,B 0,C 180,E1 -15063.918,E2 -15063.918} C_VEL
LIN {X 0,Y 343.904,Z 698.161,A -85,B 0,C 180,E1 -15065.539,E2 -15065.539} C_VEL
LIN {X 0,Y 341.471,Z 694.878,A -85,B 0,C 180,E1 -15066.614,E2 -15066.614} C_VEL
LIN {X 0,Y 338.786,Z 692.774,A -85,B 0,C 180,E1 -15067.709,E2 -15067.709} C_VEL
LIN {X 0,Y 336.627,Z 689.566,A -85,B 0,C 180,E1 -15068.643,E2 -15068.643} C_VEL
LIN {X 0,Y 333.473,Z 687.088,A -85,B 0,C 180,E1 -15069.87,E2 -15069.87} C_VEL
LIN {X 0,Y 331.536,Z 684.028,A -85,B 0,C 180,E1 -15070.689,E2 -15070.689} C_VEL
LIN {X 0,Y 331.024,Z 683.392,A -85,B 0,C 180,E1 -15070.891,E2 -15070.891} C_VEL
LIN {X 0,Y 328.474,Z 681.602,A -85,B 0,C 180,E1 -15071.857,E2 -15071.857} C_VEL
LIN {X 0,Y 327.002,Z 679.132,A -85,B 0,C 180,E1 -15072.473,E2 -15072.473} C_VEL
LIN {X 0,Y 326.667,Z 677.977,A -85,B 0,C 180,E1 -15072.861,E2 -15072.861} C_VEL
LIN {X 0,Y 326.603,Z 677.64,A -85,B 0,C 180,E1 -15073.517,E2 -15073.517} C_VEL
LIN {X 0,Y 326.621,Z 677.615,A -85,B 0,C 180,E1 -15077.018,E2 -15077.018} C_VEL
LIN {X 0,Y 326.638,Z 677.611,A -85,B 0,C 180,E1 -15080.765,E2 -15080.765} C_VEL
LIN {X 0,Y 326.604,Z 677.565,A -85,B 0,C 180,E1 -15084.48,E2 -15084.48} C_VEL
LIN {X 0,Y 326.6,Z 677.618,A -85,B 0,C 180,E1 -15087.455,E2 -15087.455} C_VEL
LIN {X 0,Y 326.653,Z 677.551,A -85,B 0,C 180,E1 -15090.341,E2 -15090.341} C_VEL
LIN {X 0,Y 326.684,Z 677.597,A -85,B 0,C 180,E1 -15094.516,E2 -15094.516} C_VEL
LIN {X 0,Y 326.658,Z 677.596,A -85,B 0,C 180,E1 -15098.547,E2 -15098.547} C_VEL
LIN {X 0,Y 326.736,Z 677.587,A -85,B 0,C 180,E1 -15101.178,E2 -15101.178} C_VEL
LIN {X 0,Y 326.749,Z 677.591,A -85,B 0,C 180,E1 -15105.28,E2 -15105.28} C_VEL
LIN {X 0,Y 326.099,Z 677.67,A -85,B 0,C 180,E1 -15106.309,E2 -15106.309} C_VEL
LIN {X 0,Y 323.235,Z 678.029,A -85,B 0,C 180,E1 -15107.983,E2 -15107.983} C_VEL
LIN {X 0,Y 320.827,Z 678.33,A -85,B 0,C 180,E1 -15109.34,E2 -15109.34} C_VEL
LIN {X 0,Y 319.842,Z 678.449,A -85,B 0,C 180,E1 -15110.391,E2 -15110.391} C_VEL
LIN {X 0,Y 319.788,Z 678.45,A -85,B 0,C 180,E1 -15110.747,E2 -15110.747} C_VEL
LIN {X 0,Y 319.94,Z 678.435,A -85,B 0,C 180,E1 -15113.695,E2 -15113.695} C_VEL
LIN {X 0,Y 319.984,Z 678.416,A -85,B 0,C 180,E1 -15117.483,E2 -15117.483} C_VEL
LIN {X 0,Y 320.161,Z 678.417,A -85,B 0,C 180,E1 -15120,E2 -15120} C_VEL
LIN {X 0,Y 319.984,Z 678.418,A -85,B 0,C 180,E1 -15122.518,E2 -15122.518} C_VEL
LIN {X 0,Y 319.941,Z 678.436,A -85,B 0,C 180,E1 -15126.306,E2 -15126.306} C_VEL
LIN {X 0,Y 319.835,Z 678.437,A -85,B 0,C 180,E1 -15128.848,E2 -15128.848} C_VEL
LIN {X 0,Y 319.677,Z 678.456,A -85,B 0,C 180,E1 -15132.7,E2 -15132.7} C_VEL
LIN {X 0,Y 319.692,Z 678.474,A -85,B 0,C 180,E1 -15135.296,E2 -15135.296} C_VEL
LIN {X 0,Y 319.67,Z 678.47,A -85,B 0,C 180,E1 -15139.255,E2 -15139.255} C_VEL
LIN {X 0,Y 319.564,Z 678.478,A -85,B 0,C 180,E1 -15143.32,E2 -15143.32} C_VEL
LIN {X 0,Y 319.629,Z 678.461,A -85,B 0,C 180,E1 -15146.089,E2 -15146.089} C_VEL
LIN {X 0,Y 319.583,Z 678.423,A -85,B 0,C 180,E1 -15148.934,E2 -15148.934} C_VEL
LIN {X 0,Y 319.526,Z 678.487,A -85,B 0,C 180,E1 -15151.863,E2 -15151.863} C_VEL
LIN {X 0,Y 319.574,Z 678.449,A -85,B 0,C 180,E1 -15155.544,E2 -15155.544} C_VEL
LIN {X 0,Y 319.596,Z 678.476,A -85,B 0,C 180,E1 -15158.005,E2 -15158.005} C_VEL
LIN {X 0,Y 319.611,Z 678.587,A -85,B 0,C 180,E1 -15160.961,E2 -15160.961} C_VEL
LIN {X 0,Y 322.123,Z 686.649,A -85,B 0,C 180,E1 -15164.06,E2 -15164.06} C_VEL
LIN {X 0,Y 322.566,Z 687.846,A -85,B 0,C 180,E1 -15164.367,E2 -15164.367} C_VEL
LIN {X 0,Y 325.366,Z 692.453,A -85,B 0,C 180,E1 -15165.025,E2 -15165.025} C_VEL
LIN {X 0,Y 334.701,Z 708.318,A -85,B 0,C 180,E1 -15167.045,E2 -15167.045} C_VEL
LIN {X 0,Y 342.142,Z 722.27,A -85,B 0,C 180,E1 -15168.569,E2 -15168.569} C_VEL
LIN {X 0,Y 350.494,Z 739.372,A -85,B 0,C 180,E1 -15170.202,E2 -15170.202} C_VEL
LIN {X 0,Y 353.246,Z 746.067,A -85,B 0,C 180,E1 -15170.742,E2 -15170.742} C_VEL
LIN {X 0,Y 354.269,Z 751.211,A -85,B 0,C 180,E1 -15171.007,E2 -15171.007} C_VEL
LIN {X 0,Y 348.901,Z 891.79,A -85,B 0,C 180,E1 -15173.919,E2 -15173.919} C_VEL
LIN {X 0,Y 348.167,Z 902.437,A -85,B 0,C 180,E1 -15174.215,E2 -15174.215} C_VEL
LIN {X 0,Y 346.668,Z 916.749,A -85,B 0,C 180,E1 -15174.751,E2 -15174.751} C_VEL
LIN {X 0,Y 345.003,Z 929.865,A -85,B 0,C 180,E1 -15175.402,E2 -15175.402} C_VEL
LIN {X 0,Y 343.432,Z 941.253,A -85,B 0,C 180,E1 -15176.108,E2 -15176.108} C_VEL
LIN {X 0,Y 341.146,Z 954.486,A -85,B 0,C 180,E1 -15177.089,E2 -15177.089} C_VEL
LIN {X 0,Y 338.908,Z 966.647,A -85,B 0,C 180,E1 -15178.181,E2 -15178.181} C_VEL
LIN {X 0,Y 336.525,Z 978.22,A -85,B 0,C 180,E1 -15179.4,E2 -15179.4} C_VEL
LIN {X 0,Y 334.081,Z 989.018,A -85,B 0,C 180,E1 -15180.719,E2 -15180.719} C_VEL
LIN {X 0,Y 331.681,Z 999.518,A -85,B 0,C 180,E1 -15182.216,E2 -15182.216} C_VEL
LIN {X 0,Y 329.354,Z 1009.137,A -85,B 0,C 180,E1 -15183.791,E2 -15183.791} C_VEL
LIN {X 0,Y 327.053,Z 1018.52,A -85,B 0,C 180,E1 -15185.566,E2 -15185.566} C_VEL
LIN {X 0,Y 324.987,Z 1027.046,A -85,B 0,C 180,E1 -15187.428,E2 -15187.428} C_VEL
LIN {X 0,Y 322.983,Z 1035.649,A -85,B 0,C 180,E1 -15189.626,E2 -15189.626} C_VEL
LIN {X 0,Y 321.57,Z 1042.082,A -85,B 0,C 180,E1 -15191.525,E2 -15191.525} C_VEL
LIN {X 0,Y 320.004,Z 1049.344,A -85,B 0,C 180,E1 -15194.067,E2 -15194.067} C_VEL
LIN {X 0,Y 319.233,Z 1053.999,A -85,B 0,C 180,E1 -15195.986,E2 -15195.986} C_VEL
LIN {X 0,Y 318.432,Z 1059.098,A -85,B 0,C 180,E1 -15198.543,E2 -15198.543} C_VEL
LIN {X 0,Y 317.994,Z 1063.099,A -85,B 0,C 180,E1 -15201.1,E2 -15201.1} C_VEL
LIN {X 0,Y 317.851,Z 1066.057,A -85,B 0,C 180,E1 -15203.653,E2 -15203.653} C_VEL
LIN {X 0,Y 317.768,Z 1067.243,A -85,B 0,C 180,E1 -15204.925,E2 -15204.925} C_VEL
LIN {X 0,Y 317.742,Z 1068.711,A -85,B 0,C 180,E1 -15207.465,E2 -15207.465} C_VEL
LIN {X 0,Y 317.779,Z 1069.199,A -85,B 0,C 180,E1 -15210,E2 -15210} C_VEL
LIN {X 0,Y 317.742,Z 1068.711,A -85,B 0,C 180,E1 -15212.535,E2 -15212.535} C_VEL
LIN {X 0,Y 317.808,Z 1066.699,A -85,B 0,C 180,E1 -15215.659,E2 -15215.659} C_VEL
LIN {X 0,Y 317.865,Z 1064.773,A -85,B 0,C 180,E1 -15217.623,E2 -15217.623} C_VEL
LIN {X 0,Y 318.263,Z 1060.186,A -85,B 0,C 180,E1 -15220.818,E2 -15220.818} C_VEL
LIN {X 0,Y 318.782,Z 1056.697,A -85,B 0,C 180,E1 -15222.736,E2 -15222.736} C_VEL
LIN {X 0,Y 319.529,Z 1052.282,A -85,B 0,C 180,E1 -15224.775,E2 -15224.775} C_VEL
LIN {X 0,Y 320.706,Z 1045.905,A -85,B 0,C 180,E1 -15227.208,E2 -15227.208} C_VEL
LIN {X 0,Y 322.504,Z 1037.873,A -85,B 0,C 180,E1 -15229.741,E2 -15229.741} C_VEL
LIN {X 0,Y 324.031,Z 1030.885,A -85,B 0,C 180,E1 -15231.636,E2 -15231.636} C_VEL
LIN {X 0,Y 326.003,Z 1022.917,A -85,B 0,C 180,E1 -15233.504,E2 -15233.504} C_VEL
LIN {X 0,Y 328.299,Z 1013.806,A -85,B 0,C 180,E1 -15235.349,E2 -15235.349} C_VEL
LIN {X 0,Y 330.298,Z 1005.235,A -85,B 0,C 180,E1 -15236.881,E2 -15236.881} C_VEL
LIN {X 0,Y 333.128,Z 993.371,A -85,B 0,C 180,E1 -15238.682,E2 -15238.682} C_VEL
LIN {X 0,Y 335.347,Z 983.204,A -85,B 0,C 180,E1 -15240.023,E2 -15240.023} C_VEL
LIN {X 0,Y 337.89,Z 971.537,A -85,B 0,C 180,E1 -15241.331,E2 -15241.331} C_VEL
LIN {X 0,Y 340.255,Z 959.513,A -85,B 0,C 180,E1 -15242.481,E2 -15242.481} C_VEL
LIN {X 0,Y 342.441,Z 947.195,A -85,B 0,C 180,E1 -15243.473,E2 -15243.473} C_VEL
LIN {X 0,Y 344.416,Z 934.654,A -85,B 0,C 180,E1 -15244.311,E2 -15244.311} C_VEL
LIN {X 0,Y 345.997,Z 921.97,A -85,B 0,C 180,E1 -15245.016,E2 -15245.016} C_VEL
LIN {X 0,Y 347.579,Z 908.31,A -85,B 0,C 180,E1 -15245.587,E2 -15245.587} C_VEL
LIN {X 0,Y 348.729,Z 895.152,A -85,B 0,C 180,E1 -15245.995,E2 -15245.995} C_VEL
LIN {X 0,Y 349.802,Z 869.848,A -85,B 0,C 180,E1 -15246.561,E2 -15246.561} C_VEL
LIN {X 0,Y 354.23,Z 750.748,A -85,B 0,C 180,E1 -15249.01,E2 -15249.01} C_VEL
LIN {X 0,Y 352.835,Z 744.714,A -85,B 0,C 180,E1 -15249.347,E2 -15249.347} C_VEL
LIN {X 0,Y 346.472,Z 730.826,A -85,B 0,C 180,E1 -15250.578,E2 -15250.578} C_VEL
LIN {X 0,Y 336.623,Z 711.699,A -85,B 0,C 180,E1 -15252.558,E2 -15252.558} C_VEL
LIN {X 0,Y 327.965,Z 696.823,A -85,B 0,C 180,E1 -15254.396,E2 -15254.396} C_VEL
LIN {X 0,Y 322.471,Z 687.588,A -85,B 0,C 180,E1 -15255.671,E2 -15255.671} C_VEL
LIN {X 0,Y 320.465,Z 681.359,A -85,B 0,C 180,E1 -15257.903,E2 -15257.903} C_VEL
LIN {X 0,Y 319.585,Z 678.545,A -85,B 0,C 180,E1 -15259.087,E2 -15259.087} C_VEL
LIN {X 0,Y 319.594,Z 678.468,A -85,B 0,C 180,E1 -15262.338,E2 -15262.338} C_VEL
LIN {X 0,Y 319.554,Z 678.456,A -85,B 0,C 180,E1 -15265.123,E2 -15265.123} C_VEL
LIN {X 0,Y 319.564,Z 678.454,A -85,B 0,C 180,E1 -15269.057,E2 -15269.057} C_VEL
LIN {X 0,Y 319.602,Z 678.43,A -85,B 0,C 180,E1 -15272.497,E2 -15272.497} C_VEL
LIN {X 0,Y 319.599,Z 678.487,A -85,B 0,C 180,E1 -15275.303,E2 -15275.303} C_VEL
LIN {X 0,Y 319.592,Z 678.471,A -85,B 0,C 180,E1 -15278.047,E2 -15278.047} C_VEL
LIN {X 0,Y 319.684,Z 678.466,A -85,B 0,C 180,E1 -15280.961,E2 -15280.961} C_VEL
LIN {X 0,Y 319.724,Z 678.467,A -85,B 0,C 180,E1 -15285.275,E2 -15285.275} C_VEL
LIN {X 0,Y 319.751,Z 678.465,A -85,B 0,C 180,E1 -15289.872,E2 -15289.872} C_VEL
LIN {X 0,Y 319.92,Z 678.423,A -85,B 0,C 180,E1 -15292.426,E2 -15292.426} C_VEL
LIN {X 0,Y 319.743,Z 678.467,A -85,B 0,C 180,E1 -15294.956,E2 -15294.956} C_VEL
LIN {X 0,Y 319.984,Z 678.417,A -85,B 0,C 180,E1 -15297.482,E2 -15297.482} C_VEL
LIN {X 0,Y 320.161,Z 678.415,A -85,B 0,C 180,E1 -15300,E2 -15300} C_VEL
LIN {X 0,Y 319.984,Z 678.415,A -85,B 0,C 180,E1 -15302.517,E2 -15302.517} C_VEL
LIN {X 0,Y 319.922,Z 678.435,A -85,B 0,C 180,E1 -15306.577,E2 -15306.577} C_VEL
LIN {X 0,Y 319.834,Z 678.444,A -85,B 0,C 180,E1 -15308.848,E2 -15308.848} C_VEL
LIN {X 0,Y 319.672,Z 678.455,A -85,B 0,C 180,E1 -15312.7,E2 -15312.7} C_VEL
LIN {X 0,Y 319.691,Z 678.474,A -85,B 0,C 180,E1 -15315.295,E2 -15315.295} C_VEL
LIN {X 0,Y 319.672,Z 678.473,A -85,B 0,C 180,E1 -15319.255,E2 -15319.255} C_VEL
LIN {X 0,Y 319.569,Z 678.48,A -85,B 0,C 180,E1 -15323.319,E2 -15323.319} C_VEL
LIN {X 0,Y 319.628,Z 678.46,A -85,B 0,C 180,E1 -15326.088,E2 -15326.088} C_VEL
LIN {X 0,Y 319.581,Z 678.425,A -85,B 0,C 180,E1 -15328.934,E2 -15328.934} C_VEL
LIN {X 0,Y 319.524,Z 678.489,A -85,B 0,C 180,E1 -15331.862,E2 -15331.862} C_VEL
LIN {X 0,Y 319.572,Z 678.439,A -85,B 0,C 180,E1 -15335.543,E2 -15335.543} C_VEL
LIN {X 0,Y 319.576,Z 678.457,A -85,B 0,C 180,E1 -15338.007,E2 -15338.007} C_VEL
LIN {X 0,Y 319.59,Z 678.489,A -85,B 0,C 180,E1 -15341.612,E2 -15341.612} C_VEL
LIN {X 0,Y 319.6,Z 678.734,A -85,B 0,C 180,E1 -15344.831,E2 -15344.831} C_VEL
LIN {X 0,Y 319.932,Z 680.089,A -85,B 0,C 180,E1 -15345.284,E2 -15345.284} C_VEL
LIN {X 0,Y 321.484,Z 682.563,A -85,B 0,C 180,E1 -15345.915,E2 -15345.915} C_VEL
LIN {X 0,Y 324.351,Z 684.684,A -85,B 0,C 180,E1 -15346.903,E2 -15346.903} C_VEL
LIN {X 0,Y 326.207,Z 687.815,A -85,B 0,C 180,E1 -15347.68,E2 -15347.68} C_VEL
LIN {X 0,Y 328.795,Z 689.887,A -85,B 0,C 180,E1 -15348.648,E2 -15348.648} C_VEL
LIN {X 0,Y 329.446,Z 690.54,A -85,B 0,C 180,E1 -15348.905,E2 -15348.905} C_VEL
LIN {X 0,Y 331.733,Z 693.752,A -85,B 0,C 180,E1 -15349.831,E2 -15349.831} C_VEL
LIN {X 0,Y 334.77,Z 696.36,A -85,B 0,C 180,E1 -15351.024,E2 -15351.024} C_VEL
LIN {X 0,Y 337.341,Z 699.732,A -85,B 0,C 180,E1 -15352.116,E2 -15352.116} C_VEL
LIN {X 0,Y 340.231,Z 702.177,A -85,B 0,C 180,E1 -15353.292,E2 -15353.292} C_VEL
LIN {X 0,Y 343.053,Z 705.696,A -85,B 0,C 180,E1 -15354.522,E2 -15354.522} C_VEL
LIN {X 0,Y 346.087,Z 708.259,A -85,B 0,C 180,E1 -15355.816,E2 -15355.816} C_VEL
LIN {X 0,Y 349.104,Z 711.877,A -85,B 0,C 180,E1 -15357.2,E2 -15357.2} C_VEL
LIN {X 0,Y 352.333,Z 714.478,A -85,B 0,C 180,E1 -15358.664,E2 -15358.664} C_VEL
LIN {X 0,Y 355.295,Z 717.975,A -85,B 0,C 180,E1 -15360.119,E2 -15360.119} C_VEL
LIN {X 0,Y 358.629,Z 720.622,A -85,B 0,C 180,E1 -15361.751,E2 -15361.751} C_VEL
LIN {X 0,Y 361.318,Z 723.922,A -85,B 0,C 180,E1 -15363.196,E2 -15363.196} C_VEL
LIN {X 0,Y 364.532,Z 726.317,A -85,B 0,C 180,E1 -15364.904,E2 -15364.904} C_VEL
LIN {X 0,Y 367.791,Z 730.199,A -85,B 0,C 180,E1 -15366.877,E2 -15366.877} C_VEL
LIN {X 0,Y 370.928,Z 732.529,A -85,B 0,C 180,E1 -15368.802,E2 -15368.802} C_VEL
LIN {X 0,Y 372.207,Z 733.378,A -85,B 0,C 180,E1 -15369.64,E2 -15369.64} C_VEL
LIN {X 0,Y 374.617,Z 736.469,A -85,B 0,C 180,E1 -15371.402,E2 -15371.402} C_VEL
LIN {X 0,Y 377.514,Z 738.77,A -85,B 0,C 180,E1 -15373.639,E2 -15373.639} C_VEL
LIN {X 0,Y 379.692,Z 740.039,A -85,B 0,C 180,E1 -15375.461,E2 -15375.461} C_VEL
LIN {X 0,Y 381.51,Z 742.668,A -85,B 0,C 180,E1 -15377.4,E2 -15377.4} C_VEL
LIN {X 0,Y 383.27,Z 744.335,A -85,B 0,C 180,E1 -15379.434,E2 -15379.434} C_VEL
LIN {X 0,Y 385.086,Z 745.372,A -85,B 0,C 180,E1 -15381.93,E2 -15381.93} C_VEL
LIN {X 0,Y 386.596,Z 746.093,A -85,B 0,C 180,E1 -15384.785,E2 -15384.785} C_VEL
LIN {X 0,Y 387.252,Z 746.504,A -85,B 0,C 180,E1 -15386.879,E2 -15386.879} C_VEL
LIN {X 0,Y 387.58,Z 746.786,A -85,B 0,C 180,E1 -15388.961,E2 -15388.961} C_VEL
LIN {X 0,Y 387.58,Z 746.788,A -85,B 0,C 180,E1 -15391.039,E2 -15391.039} C_VEL
LIN {X 0,Y 387.194,Z 746.488,A -85,B 0,C 180,E1 -15393.342,E2 -15393.342} C_VEL
LIN {X 0,Y 386.292,Z 745.983,A -85,B 0,C 180,E1 -15395.813,E2 -15395.813} C_VEL
LIN {X 0,Y 384.861,Z 745.247,A -85,B 0,C 180,E1 -15398.4,E2 -15398.4} C_VEL
LIN {X 0,Y 382.983,Z 744.116,A -85,B 0,C 180,E1 -15400.903,E2 -15400.903} C_VEL
LIN {X 0,Y 381.003,Z 742.03,A -85,B 0,C 180,E1 -15403.177,E2 -15403.177} C_VEL
LIN {X 0,Y 379.453,Z 739.734,A -85,B 0,C 180,E1 -15404.754,E2 -15404.754} C_VEL
LIN {X 0,Y 376.523,Z 738.114,A -85,B 0,C 180,E1 -15407.153,E2 -15407.153} C_VEL
LIN {X 0,Y 373.851,Z 735.63,A -85,B 0,C 180,E1 -15409.161,E2 -15409.161} C_VEL
LIN {X 0,Y 372.012,Z 733.127,A -85,B 0,C 180,E1 -15410.501,E2 -15410.501} C_VEL
LIN {X 0,Y 368.52,Z 730.846,A -85,B 0,C 180,E1 -15412.683,E2 -15412.683} C_VEL
LIN {X 0,Y 365.641,Z 727.671,A -85,B 0,C 180,E1 -15414.428,E2 -15414.428} C_VEL
LIN {X 0,Y 364.532,Z 726.318,A -85,B 0,C 180,E1 -15415.096,E2 -15415.096} C_VEL
LIN {X 0,Y 361.318,Z 723.921,A -85,B 0,C 180,E1 -15416.804,E2 -15416.804} C_VEL
LIN {X 0,Y 358.629,Z 720.635,A -85,B 0,C 180,E1 -15418.249,E2 -15418.249} C_VEL
LIN {X 0,Y 354.634,Z 717.303,A -85,B 0,C 180,E1 -15420.213,E2 -15420.213} C_VEL
LIN {X 0,Y 351.635,Z 713.785,A -85,B 0,C 180,E1 -15421.673,E2 -15421.673} C_VEL
LIN {X 0,Y 348.127,Z 710.865,A -85,B 0,C 180,E1 -15423.254,E2 -15423.254} C_VEL
LIN {X 0,Y 345.357,Z 707.484,A -85,B 0,C 180,E1 -15424.518,E2 -15424.518} C_VEL
LIN {X 0,Y 342.12,Z 704.699,A -85,B 0,C 180,E1 -15425.892,E2 -15425.892} C_VEL
LIN {X 0,Y 339.692,Z 701.54,A -85,B 0,C 180,E1 -15426.941,E2 -15426.941} C_VEL
LIN {X 0,Y 336.803,Z 699.179,A -85,B 0,C 180,E1 -15428.105,E2 -15428.105} C_VEL
LIN {X 0,Y 334.162,Z 695.726,A -85,B 0,C 180,E1 -15429.215,E2 -15429.215} C_VEL
LIN {X 0,Y 331.31,Z 693.293,A -85,B 0,C 180,E1 -15430.337,E2 -15430.337} C_VEL
LIN {X 0,Y 329.18,Z 690.089,A -85,B 0,C 180,E1 -15431.209,E2 -15431.209} C_VEL
LIN {X 0,Y 326.433,Z 688.063,A -85,B 0,C 180,E1 -15432.233,E2 -15432.233} C_VEL
LIN {X 0,Y 324.574,Z 685.17,A -85,B 0,C 180,E1 -15432.998,E2 -15432.998} C_VEL
LIN {X 0,Y 324.057,Z 684.337,A -85,B 0,C 180,E1 -15433.209,E2 -15433.209} C_VEL
LIN {X 0,Y 321.329,Z 682.382,A -85,B 0,C 180,E1 -15434.142,E2 -15434.142} C_VEL
LIN {X 0,Y 319.864,Z 679.889,A -85,B 0,C 180,E1 -15434.75,E2 -15434.75} C_VEL
LIN {X 0,Y 319.57,Z 678.67,A -85,B 0,C 180,E1 -15435.218,E2 -15435.218} C_VEL
LIN {X 0,Y 319.572,Z 678.492,A -85,B 0,C 180,E1 -15438.719,E2 -15438.719} C_VEL
LIN {X 0,Y 319.575,Z 678.45,A -85,B 0,C 180,E1 -15442.343,E2 -15442.343} C_VEL
LIN {X 0,Y 319.551,Z 678.449,A -85,B 0,C 180,E1 -15445.123,E2 -15445.123} C_VEL
LIN {X 0,Y 319.562,Z 678.458,A -85,B 0,C 180,E1 -15449.058,E2 -15449.058} C_VEL
LIN {X 0,Y 319.601,Z 678.431,A -85,B 0,C 180,E1 -15452.498,E2 -15452.498} C_VEL
LIN {X 0,Y 319.604,Z 678.487,A -85,B 0,C 180,E1 -15455.305,E2 -15455.305} C_VEL
LIN {X 0,Y 319.625,Z 678.481,A -85,B 0,C 180,E1 -15459.402,E2 -15459.402} C_VEL
LIN {X 0,Y 319.65,Z 678.461,A -85,B 0,C 180,E1 -15462.073,E2 -15462.073} C_VEL
LIN {X 0,Y 319.723,Z 678.456,A -85,B 0,C 180,E1 -15466.008,E2 -15466.008} C_VEL
LIN {X 0,Y 319.749,Z 678.466,A -85,B 0,C 180,E1 -15469.873,E2 -15469.873} C_VEL
LIN {X 0,Y 319.788,Z 678.45,A -85,B 0,C 180,E1 -15470.747,E2 -15470.747} C_VEL
LIN {X 0,Y 319.51,Z 678.481,A -85,B 0,C 180,E1 -15471.45,E2 -15471.45} C_VEL
LIN {X 0,Y 317.541,Z 678.73,A -85,B 0,C 180,E1 -15472.829,E2 -15472.829} C_VEL
LIN {X 0,Y 313.744,Z 679.215,A -85,B 0,C 180,E1 -15474.894,E2 -15474.894} C_VEL
LIN {X 0,Y 312.755,Z 679.329,A -85,B 0,C 180,E1 -15475.969,E2 -15475.969} C_VEL
LIN {X 0,Y 312.717,Z 679.328,A -85,B 0,C 180,E1 -15476.333,E2 -15476.333} C_VEL
LIN {X 0,Y 312.984,Z 679.297,A -85,B 0,C 180,E1 -15478.714,E2 -15478.714} C_VEL
LIN {X 0,Y 313.113,Z 679.295,A -85,B 0,C 180,E1 -15480,E2 -15480} C_VEL
LIN {X 0,Y 312.93,Z 679.296,A -85,B 0,C 180,E1 -15482.575,E2 -15482.575} C_VEL
LIN {X 0,Y 312.899,Z 679.31,A -85,B 0,C 180,E1 -15486.448,E2 -15486.448} C_VEL
LIN {X 0,Y 312.78,Z 679.317,A -85,B 0,C 180,E1 -15489.05,E2 -15489.05} C_VEL
LIN {X 0,Y 312.629,Z 679.333,A -85,B 0,C 180,E1 -15492.992,E2 -15492.992} C_VEL
LIN {X 0,Y 312.631,Z 679.352,A -85,B 0,C 180,E1 -15495.65,E2 -15495.65} C_VEL
LIN {X 0,Y 312.6,Z 679.356,A -85,B 0,C 180,E1 -15499.709,E2 -15499.709} C_VEL
LIN {X 0,Y 312.539,Z 679.348,A -85,B 0,C 180,E1 -15502.79,E2 -15502.79} C_VEL
LIN {X 0,Y 312.597,Z 679.34,A -85,B 0,C 180,E1 -15505.936,E2 -15505.936} C_VEL
LIN {X 0,Y 312.539,Z 679.304,A -85,B 0,C 180,E1 -15509.651,E2 -15509.651} C_VEL
LIN {X 0,Y 312.514,Z 679.352,A -85,B 0,C 180,E1 -15513.69,E2 -15513.69} C_VEL
LIN {X 0,Y 312.548,Z 679.338,A -85,B 0,C 180,E1 -15517.382,E2 -15517.382} C_VEL
LIN {X 0,Y 312.552,Z 679.417,A -85,B 0,C 180,E1 -15519.811,E2 -15519.811} C_VEL
LIN {X 0,Y 313.02,Z 681.176,A -85,B 0,C 180,E1 -15520.626,E2 -15520.626} C_VEL
LIN {X 0,Y 314.957,Z 687.074,A -85,B 0,C 180,E1 -15522.888,E2 -15522.888} C_VEL
LIN {X 0,Y 318.119,Z 692.175,A -85,B 0,C 180,E1 -15523.706,E2 -15523.706} C_VEL
LIN {X 0,Y 325.301,Z 704.166,A -85,B 0,C 180,E1 -15525.369,E2 -15525.369} C_VEL
LIN {X 0,Y 332.772,Z 717.336,A -85,B 0,C 180,E1 -15526.997,E2 -15526.997} C_VEL
LIN {X 0,Y 341.347,Z 734.116,A -85,B 0,C 180,E1 -15528.776,E2 -15528.776} C_VEL
LIN {X 0,Y 347.88,Z 748.385,A -85,B 0,C 180,E1 -15530.082,E2 -15530.082} C_VEL
LIN {X 0,Y 348.725,Z 752.48,A -85,B 0,C 180,E1 -15530.304,E2 -15530.304} C_VEL
LIN {X 0,Y 343.184,Z 891.528,A -85,B 0,C 180,E1 -15533.218,E2 -15533.218} C_VEL
LIN {X 0,Y 342.337,Z 903.21,A -85,B 0,C 180,E1 -15533.555,E2 -15533.555} C_VEL
LIN {X 0,Y 340.893,Z 916.544,A -85,B 0,C 180,E1 -15534.062,E2 -15534.062} C_VEL
LIN {X 0,Y 339.175,Z 929.659,A -85,B 0,C 180,E1 -15534.72,E2 -15534.72} C_VEL
LIN {X 0,Y 337.537,Z 941.047,A -85,B 0,C 180,E1 -15535.433,E2 -15535.433} C_VEL
LIN {X 0,Y 335.156,Z 954.279,A -85,B 0,C 180,E1 -15536.423,E2 -15536.423} C_VEL
LIN {X 0,Y 332.894,Z 966.154,A -85,B 0,C 180,E1 -15537.501,E2 -15537.501} C_VEL
LIN {X 0,Y 330.356,Z 978.012,A -85,B 0,C 180,E1 -15538.766,E2 -15538.766} C_VEL
LIN {X 0,Y 327.826,Z 988.81,A -85,B 0,C 180,E1 -15540.104,E2 -15540.104} C_VEL
LIN {X 0,Y 325.342,Z 999.31,A -85,B 0,C 180,E1 -15541.626,E2 -15541.626} C_VEL
LIN {X 0,Y 322.706,Z 1009.688,A -85,B 0,C 180,E1 -15543.367,E2 -15543.367} C_VEL
LIN {X 0,Y 320.512,Z 1018.312,A -85,B 0,C 180,E1 -15545.033,E2 -15545.033} C_VEL
LIN {X 0,Y 318.354,Z 1026.837,A -85,B 0,C 180,E1 -15546.931,E2 -15546.931} C_VEL
LIN {X 0,Y 316.236,Z 1035.44,A -85,B 0,C 180,E1 -15549.171,E2 -15549.171} C_VEL
LIN {X 0,Y 314.745,Z 1041.874,A -85,B 0,C 180,E1 -15551.109,E2 -15551.109} C_VEL
LIN {X 0,Y 313.075,Z 1049.135,A -85,B 0,C 180,E1 -15553.704,E2 -15553.704} C_VEL
LIN {X 0,Y 312.231,Z 1053.79,A -85,B 0,C 180,E1 -15555.665,E2 -15555.665} C_VEL
LIN {X 0,Y 311.419,Z 1058.891,A -85,B 0,C 180,E1 -15558.282,E2 -15558.282} C_VEL
LIN {X 0,Y 310.918,Z 1062.892,A -85,B 0,C 180,E1 -15560.896,E2 -15560.896} C_VEL
LIN {X 0,Y 310.763,Z 1065.851,A -85,B 0,C 180,E1 -15563.507,E2 -15563.507} C_VEL
LIN {X 0,Y 310.683,Z 1067.037,A -85,B 0,C 180,E1 -15564.809,E2 -15564.809} C_VEL
LIN {X 0,Y 310.664,Z 1068.506,A -85,B 0,C 180,E1 -15567.407,E2 -15567.407} C_VEL
LIN {X 0,Y 310.689,Z 1068.994,A -85,B 0,C 180,E1 -15570,E2 -15570} C_VEL
LIN {X 0,Y 310.664,Z 1068.506,A -85,B 0,C 180,E1 -15572.593,E2 -15572.593} C_VEL
LIN {X 0,Y 310.723,Z 1066.651,A -85,B 0,C 180,E1 -15575.616,E2 -15575.616} C_VEL
LIN {X 0,Y 310.784,Z 1064.567,A -85,B 0,C 180,E1 -15577.798,E2 -15577.798} C_VEL
LIN {X 0,Y 311.239,Z 1059.979,A -85,B 0,C 180,E1 -15581.066,E2 -15581.066} C_VEL
LIN {X 0,Y 311.771,Z 1056.488,A -85,B 0,C 180,E1 -15583.027,E2 -15583.027} C_VEL
LIN {X 0,Y 312.763,Z 1050.758,A -85,B 0,C 180,E1 -15585.643,E2 -15585.643} C_VEL
LIN {X 0,Y 313.822,Z 1045.696,A -85,B 0,C 180,E1 -15587.597,E2 -15587.597} C_VEL
LIN {X 0,Y 315.694,Z 1037.663,A -85,B 0,C 180,E1 -15590.185,E2 -15590.185} C_VEL
LIN {X 0,Y 317.324,Z 1030.676,A -85,B 0,C 180,E1 -15592.117,E2 -15592.117} C_VEL
LIN {X 0,Y 319.403,Z 1022.709,A -85,B 0,C 180,E1 -15594.02,E2 -15594.02} C_VEL
LIN {X 0,Y 321.789,Z 1013.597,A -85,B 0,C 180,E1 -15595.9,E2 -15595.9} C_VEL
LIN {X 0,Y 323.9,Z 1005.027,A -85,B 0,C 180,E1 -15597.456,E2 -15597.456} C_VEL
LIN {X 0,Y 326.859,Z 993.164,A -85,B 0,C 180,E1 -15599.285,E2 -15599.285} C_VEL
LIN {X 0,Y 329.178,Z 982.997,A -85,B 0,C 180,E1 -15600.645,E2 -15600.645} C_VEL
LIN {X 0,Y 331.8,Z 971.33,A -85,B 0,C 180,E1 -15601.973,E2 -15601.973} C_VEL
LIN {X 0,Y 334.232,Z 959.306,A -85,B 0,C 180,E1 -15603.141,E2 -15603.141} C_VEL
LIN {X 0,Y 336.509,Z 946.989,A -85,B 0,C 180,E1 -15604.144,E2 -15604.144} C_VEL
LIN {X 0,Y 338.543,Z 934.447,A -85,B 0,C 180,E1 -15604.992,E2 -15604.992} C_VEL
LIN {X 0,Y 340.28,Z 921.018,A -85,B 0,C 180,E1 -15605.739,E2 -15605.739} C_VEL
LIN {X 0,Y 341.822,Z 908.104,A -85,B 0,C 180,E1 -15606.28,E2 -15606.28} C_VEL
LIN {X 0,Y 343.041,Z 894.739,A -85,B 0,C 180,E1 -15606.695,E2 -15606.695} C_VEL
LIN {X 0,Y 344.137,Z 869.084,A -85,B 0,C 180,E1 -15607.278,E2 -15607.278} C_VEL
LIN {X 0,Y 348.679,Z 753.069,A -85,B 0,C 180,E1 -15609.687,E2 -15609.687} C_VEL
LIN {X 0,Y 347.74,Z 748.077,A -85,B 0,C 180,E1 -15609.945,E2 -15609.945} C_VEL
LIN {X 0,Y 341.615,Z 734.601,A -85,B 0,C 180,E1 -15611.171,E2 -15611.171} C_VEL
LIN {X 0,Y 332.119,Z 716.029,A -85,B 0,C 180,E1 -15613.145,E2 -15613.145} C_VEL
LIN {X 0,Y 323.727,Z 701.458,A -85,B 0,C 180,E1 -15614.987,E2 -15614.987} C_VEL
LIN {X 0,Y 317.686,Z 691.575,A -85,B 0,C 180,E1 -15616.394,E2 -15616.394} C_VEL
LIN {X 0,Y 314.968,Z 687.048,A -85,B 0,C 180,E1 -15617.113,E2 -15617.113} C_VEL
LIN {X 0,Y 312.589,Z 679.715,A -85,B 0,C 180,E1 -15619.979,E2 -15619.979} C_VEL
LIN {X 0,Y 312.547,Z 679.348,A -85,B 0,C 180,E1 -15620.403,E2 -15620.403} C_VEL
LIN {X 0,Y 312.527,Z 679.325,A -85,B 0,C 180,E1 -15624.22,E2 -15624.22} C_VEL
LIN {X 0,Y 312.499,Z 679.373,A -85,B 0,C 180,E1 -15627.333,E2 -15627.333} C_VEL
LIN {X 0,Y 312.545,Z 679.298,A -85,B 0,C 180,E1 -15631.276,E2 -15631.276} C_VEL
LIN {X 0,Y 312.579,Z 679.357,A -85,B 0,C 180,E1 -15634.71,E2 -15634.71} C_VEL
LIN {X 0,Y 312.581,Z 679.342,A -85,B 0,C 180,E1 -15637.528,E2 -15637.528} C_VEL
LIN {X 0,Y 312.632,Z 679.337,A -85,B 0,C 180,E1 -15641.656,E2 -15641.656} C_VEL
LIN {X 0,Y 312.687,Z 679.338,A -85,B 0,C 180,E1 -15645.686,E2 -15645.686} C_VEL
LIN {X 0,Y 312.696,Z 679.345,A -85,B 0,C 180,E1 -15649.641,E2 -15649.641} C_VEL
LIN {X 0,Y 312.86,Z 679.301,A -85,B 0,C 180,E1 -15652.254,E2 -15652.254} C_VEL
LIN {X 0,Y 312.713,Z 679.344,A -85,B 0,C 180,E1 -15654.842,E2 -15654.842} C_VEL
LIN {X 0,Y 312.984,Z 679.301,A -85,B 0,C 180,E1 -15658.713,E2 -15658.713} C_VEL
LIN {X 0,Y 313.113,Z 679.293,A -85,B 0,C 180,E1 -15660,E2 -15660} C_VEL
LIN {X 0,Y 312.931,Z 679.293,A -85,B 0,C 180,E1 -15662.574,E2 -15662.574} C_VEL
LIN {X 0,Y 312.888,Z 679.31,A -85,B 0,C 180,E1 -15666.558,E2 -15666.558} C_VEL
LIN {X 0,Y 312.779,Z 679.325,A -85,B 0,C 180,E1 -15669.049,E2 -15669.049} C_VEL
LIN {X 0,Y 312.625,Z 679.332,A -85,B 0,C 180,E1 -15672.991,E2 -15672.991} C_VEL
LIN {X 0,Y 312.63,Z 679.354,A -85,B 0,C 180,E1 -15675.65,E2 -15675.65} C_VEL
LIN {X 0,Y 312.603,Z 679.356,A -85,B 0,C 180,E1 -15679.708,E2 -15679.708} C_VEL
LIN {X 0,Y 312.542,Z 679.35,A -85,B 0,C 180,E1 -15682.791,E2 -15682.791} C_VEL
LIN {X 0,Y 312.596,Z 679.339,A -85,B 0,C 180,E1 -15685.936,E2 -15685.936} C_VEL
LIN {X 0,Y 312.537,Z 679.306,A -85,B 0,C 180,E1 -15689.65,E2 -15689.65} C_VEL
LIN {X 0,Y 312.512,Z 679.351,A -85,B 0,C 180,E1 -15693.689,E2 -15693.689} C_VEL
LIN {X 0,Y 312.534,Z 679.321,A -85,B 0,C 180,E1 -15697.383,E2 -15697.383} C_VEL
LIN {X 0,Y 312.519,Z 679.37,A -85,B 0,C 180,E1 -15700.704,E2 -15700.704} C_VEL
LIN {X 0,Y 312.591,Z 679.574,A -85,B 0,C 180,E1 -15702.852,E2 -15702.852} C_VEL
LIN {X 0,Y 312.861,Z 680.736,A -85,B 0,C 180,E1 -15703.246,E2 -15703.246} C_VEL
LIN {X 0,Y 314.308,Z 683.266,A -85,B 0,C 180,E1 -15703.8,E2 -15703.8} C_VEL
LIN {X 0,Y 316.94,Z 685.421,A -85,B 0,C 180,E1 -15704.643,E2 -15704.643} C_VEL
LIN {X 0,Y 318.903,Z 688.459,A -85,B 0,C 180,E1 -15705.353,E2 -15705.353} C_VEL
LIN {X 0,Y 321.662,Z 690.747,A -85,B 0,C 180,E1 -15706.332,E2 -15706.332} C_VEL
LIN {X 0,Y 324.502,Z 694.599,A -85,B 0,C 180,E1 -15707.422,E2 -15707.422} C_VEL
LIN {X 0,Y 327.462,Z 697.156,A -85,B 0,C 180,E1 -15708.529,E2 -15708.529} C_VEL
LIN {X 0,Y 330.216,Z 700.705,A -85,B 0,C 180,E1 -15709.641,E2 -15709.641} C_VEL
LIN {X 0,Y 332.818,Z 702.948,A -85,B 0,C 180,E1 -15710.662,E2 -15710.662} C_VEL
LIN {X 0,Y 335.374,Z 706.168,A -85,B 0,C 180,E1 -15711.722,E2 -15711.722} C_VEL
LIN {X 0,Y 338.488,Z 708.904,A -85,B 0,C 180,E1 -15712.979,E2 -15712.979} C_VEL
LIN {X 0,Y 341.472,Z 712.444,A -85,B 0,C 180,E1 -15714.258,E2 -15714.258} C_VEL
LIN {X 0,Y 344.381,Z 714.911,A -85,B 0,C 180,E1 -15715.489,E2 -15715.489} C_VEL
LIN {X 0,Y 347.687,Z 718.701,A -85,B 0,C 180,E1 -15716.985,E2 -15716.985} C_VEL
LIN {X 0,Y 350.686,Z 721.121,A -85,B 0,C 180,E1 -15718.332,E2 -15718.332} C_VEL
LIN {X 0,Y 354.156,Z 725.05,A -85,B 0,C 180,E1 -15720.024,E2 -15720.024} C_VEL
LIN {X 0,Y 357.189,Z 727.475,A -85,B 0,C 180,E1 -15721.502,E2 -15721.502} C_VEL
LIN {X 0,Y 359.963,Z 730.755,A -85,B 0,C 180,E1 -15722.976,E2 -15722.976} C_VEL
LIN {X 0,Y 362.96,Z 733.039,A -85,B 0,C 180,E1 -15724.564,E2 -15724.564} C_VEL
LIN {X 0,Y 364.017,Z 734.06,A -85,B 0,C 180,E1 -15725.15,E2 -15725.15} C_VEL
LIN {X 0,Y 366.851,Z 737.344,A -85,B 0,C 180,E1 -15726.861,E2 -15726.861} C_VEL
LIN {X 0,Y 369.762,Z 739.458,A -85,B 0,C 180,E1 -15728.642,E2 -15728.642} C_VEL
LIN {X 0,Y 371.106,Z 740.439,A -85,B 0,C 180,E1 -15729.512,E2 -15729.512} C_VEL
LIN {X 0,Y 373.433,Z 743.32,A -85,B 0,C 180,E1 -15731.199,E2 -15731.199} C_VEL
LIN {X 0,Y 376.388,Z 745.693,A -85,B 0,C 180,E1 -15733.441,E2 -15733.441} C_VEL
LIN {X 0,Y 378.572,Z 746.919,A -85,B 0,C 180,E1 -15735.257,E2 -15735.257} C_VEL
LIN {X 0,Y 380.265,Z 749.353,A -85,B 0,C 180,E1 -15736.982,E2 -15736.982} C_VEL
LIN {X 0,Y 382.084,Z 751.17,A -85,B 0,C 180,E1 -15739.072,E2 -15739.072} C_VEL
LIN {X 0,Y 383.975,Z 752.31,A -85,B 0,C 180,E1 -15741.58,E2 -15741.58} C_VEL
LIN {X 0,Y 385.419,Z 753.018,A -85,B 0,C 180,E1 -15744.173,E2 -15744.173} C_VEL
LIN {X 0,Y 386.075,Z 753.466,A -85,B 0,C 180,E1 -15745.824,E2 -15745.824} C_VEL
LIN {X 0,Y 386.681,Z 753.733,A -85,B 0,C 180,E1 -15748.426,E2 -15748.426} C_VEL
LIN {X 0,Y 386.717,Z 753.81,A -85,B 0,C 180,E1 -15751.041,E2 -15751.041} C_VEL
LIN {X 0,Y 386.387,Z 753.54,A -85,B 0,C 180,E1 -15753.128,E2 -15753.128} C_VEL
LIN {X 0,Y 385.719,Z 753.153,A -85,B 0,C 180,E1 -15755.227,E2 -15755.227} C_VEL
LIN {X 0,Y 384.2,Z 752.437,A -85,B 0,C 180,E1 -15758.09,E2 -15758.09} C_VEL
LIN {X 0,Y 382.273,Z 751.307,A -85,B 0,C 180,E1 -15760.709,E2 -15760.709} C_VEL
LIN {X 0,Y 380.263,Z 749.363,A -85,B 0,C 180,E1 -15763.018,E2 -15763.018} C_VEL
LIN {X 0,Y 378.19,Z 746.609,A -85,B 0,C 180,E1 -15765.079,E2 -15765.079} C_VEL
LIN {X 0,Y 375.146,Z 744.847,A -85,B 0,C 180,E1 -15767.518,E2 -15767.518} C_VEL
LIN {X 0,Y 372.417,Z 742.132,A -85,B 0,C 180,E1 -15769.57,E2 -15769.57} C_VEL
LIN {X 0,Y 370.757,Z 740.009,A -85,B 0,C 180,E1 -15770.742,E2 -15770.742} C_VEL
LIN {X 0,Y 367.368,Z 737.796,A -85,B 0,C 180,E1 -15772.824,E2 -15772.824} C_VEL
LIN {X 0,Y 364.375,Z 734.562,A -85,B 0,C 180,E1 -15774.63,E2 -15774.63} C_VEL
LIN {X 0,Y 363.225,Z 733.193,A -85,B 0,C 180,E1 -15775.298,E2 -15775.298} C_VEL
LIN {X 0,Y 359.897,Z 730.687,A -85,B 0,C 180,E1 -15777.061,E2 -15777.061} C_VEL
LIN {X 0,Y 357.118,Z 727.346,A -85,B 0,C 180,E1 -15778.539,E2 -15778.539} C_VEL
LIN {X 0,Y 353.063,Z 723.962,A -85,B 0,C 180,E1 -15780.513,E2 -15780.513} C_VEL
LIN {X 0,Y 350.26,Z 720.649,A -85,B 0,C 180,E1 -15781.867,E2 -15781.867} C_VEL
LIN {X 0,Y 346.527,Z 717.586,A -85,B 0,C 180,E1 -15783.524,E2 -15783.524} C_VEL
LIN {X 0,Y 343.572,Z 714.121,A -85,B 0,C 180,E1 -15784.855,E2 -15784.855} C_VEL
LIN {X 0,Y 340.282,Z 711.23,A -85,B 0,C 180,E1 -15786.243,E2 -15786.243} C_VEL
LIN {X 0,Y 337.877,Z 708.16,A -85,B 0,C 180,E1 -15787.289,E2 -15787.289} C_VEL
LIN {X 0,Y 334.596,Z 705.309,A -85,B 0,C 180,E1 -15788.607,E2 -15788.607} C_VEL
LIN {X 0,Y 332.169,Z 702.241,A -85,B 0,C 180,E1 -15789.6,E2 -15789.6} C_VEL
LIN {X 0,Y 329.282,Z 699.734,A -85,B 0,C 180,E1 -15790.719,E2 -15790.719} C_VEL
LIN {X 0,Y 326.981,Z 696.529,A -85,B 0,C 180,E1 -15791.665,E2 -15791.665} C_VEL
LIN {X 0,Y 324.194,Z 694.258,A -85,B 0,C 180,E1 -15792.699,E2 -15792.699} C_VEL
LIN {X 0,Y 322.025,Z 691.063,A -85,B 0,C 180,E1 -15793.54,E2 -15793.54} C_VEL
LIN {X 0,Y 318.779,Z 688.322,A -85,B 0,C 180,E1 -15794.693,E2 -15794.693} C_VEL
LIN {X 0,Y 316.518,Z 684.919,A -85,B 0,C 180,E1 -15795.496,E2 -15795.496} C_VEL
LIN {X 0,Y 314.153,Z 683.075,A -85,B 0,C 180,E1 -15796.253,E2 -15796.253} C_VEL
LIN {X 0,Y 312.858,Z 680.721,A -85,B 0,C 180,E1 -15796.754,E2 -15796.754} C_VEL
LIN {X 0,Y 312.573,Z 679.469,A -85,B 0,C 180,E1 -15797.228,E2 -15797.228} C_VEL
LIN {X 0,Y 312.526,Z 679.362,A -85,B 0,C 180,E1 -15800.976,E2 -15800.976} C_VEL
LIN {X 0,Y 312.524,Z 679.314,A -85,B 0,C 180,E1 -15804.22,E2 -15804.22} C_VEL
LIN {X 0,Y 312.497,Z 679.375,A -85,B 0,C 180,E1 -15807.334,E2 -15807.334} C_VEL
LIN {X 0,Y 312.544,Z 679.3,A -85,B 0,C 180,E1 -15811.276,E2 -15811.276} C_VEL
LIN {X 0,Y 312.581,Z 679.356,A -85,B 0,C 180,E1 -15814.711,E2 -15814.711} C_VEL
LIN {X 0,Y 312.582,Z 679.344,A -85,B 0,C 180,E1 -15817.529,E2 -15817.529} C_VEL
LIN {X 0,Y 312.631,Z 679.337,A -85,B 0,C 180,E1 -15821.656,E2 -15821.656} C_VEL
LIN {X 0,Y 312.685,Z 679.337,A -85,B 0,C 180,E1 -15825.686,E2 -15825.686} C_VEL
LIN {X 0,Y 312.693,Z 679.344,A -85,B 0,C 180,E1 -15829.642,E2 -15829.642} C_VEL
LIN {X 0,Y 312.853,Z 679.304,A -85,B 0,C 180,E1 -15832.254,E2 -15832.254} C_VEL
LIN {X 0,Y 312.712,Z 679.344,A -85,B 0,C 180,E1 -15834.843,E2 -15834.843} C_VEL
LIN {X 0,Y 312.717,Z 679.328,A -85,B 0,C 180,E1 -15836.333,E2 -15836.333} C_VEL
LIN {X 0,Y 312.185,Z 679.39,A -85,B 0,C 180,E1 -15837.412,E2 -15837.412} C_VEL
LIN {X 0,Y 309.45,Z 679.744,A -85,B 0,C 180,E1 -15839.17,E2 -15839.17} C_VEL
LIN {X 0,Y 307.046,Z 680.049,A -85,B 0,C 180,E1 -15840.595,E2 -15840.595} C_VEL
LIN {X 0,Y 305.987,Z 680.167,A -85,B 0,C 180,E1 -15841.697,E2 -15841.697} C_VEL
LIN {X 0,Y 305.89,Z 680.175,A -85,B 0,C 180,E1 -15842.071,E2 -15842.071} C_VEL
LIN {X 0,Y 305.842,Z 680.185,A -85,B 0,C 180,E1 -15846.598,E2 -15846.598} C_VEL
LIN {X 0,Y 305.729,Z 680.198,A -85,B 0,C 180,E1 -15849.26,E2 -15849.26} C_VEL
LIN {X 0,Y 305.583,Z 680.21,A -85,B 0,C 180,E1 -15853.297,E2 -15853.297} C_VEL
LIN {X 0,Y 305.587,Z 680.228,A -85,B 0,C 180,E1 -15856.021,E2 -15856.021} C_VEL
LIN {X 0,Y 305.574,Z 680.228,A -85,B 0,C 180,E1 -15859.448,E2 -15859.448} C_VEL
LIN {X 0,Y 305.484,Z 680.228,A -85,B 0,C 180,E1 -15863.042,E2 -15863.042} C_VEL
LIN {X 0,Y 305.526,Z 680.209,A -85,B 0,C 180,E1 -15866.222,E2 -15866.222} C_VEL
LIN {X 0,Y 305.489,Z 680.176,A -85,B 0,C 180,E1 -15869.05,E2 -15869.05} C_VEL
LIN {X 0,Y 305.439,Z 680.24,A -85,B 0,C 180,E1 -15871.953,E2 -15871.953} C_VEL
LIN {X 0,Y 305.457,Z 680.207,A -85,B 0,C 180,E1 -15875.114,E2 -15875.114} C_VEL
LIN {X 0,Y 305.493,Z 680.276,A -85,B 0,C 180,E1 -15878.638,E2 -15878.638} C_VEL
LIN {X 0,Y 306.734,Z 684.317,A -85,B 0,C 180,E1 -15880.462,E2 -15880.462} C_VEL
LIN {X 0,Y 307.68,Z 687.012,A -85,B 0,C 180,E1 -15881.447,E2 -15881.447} C_VEL
LIN {X 0,Y 310.832,Z 691.875,A -85,B 0,C 180,E1 -15882.282,E2 -15882.282} C_VEL
LIN {X 0,Y 318.402,Z 704.199,A -85,B 0,C 180,E1 -15884.14,E2 -15884.14} C_VEL
LIN {X 0,Y 326.486,Z 718.256,A -85,B 0,C 180,E1 -15885.995,E2 -15885.995} C_VEL
LIN {X 0,Y 333.577,Z 731.922,A -85,B 0,C 180,E1 -15887.542,E2 -15887.542} C_VEL
LIN {X 0,Y 341.065,Z 747.659,A -85,B 0,C 180,E1 -15889.104,E2 -15889.104} C_VEL
LIN {X 0,Y 343.018,Z 752.722,A -85,B 0,C 180,E1 -15889.521,E2 -15889.521} C_VEL
LIN {X 0,Y 343.108,Z 756.742,A -85,B 0,C 180,E1 -15889.641,E2 -15889.641} C_VEL
LIN {X 0,Y 337.53,Z 891.152,A -85,B 0,C 180,E1 -15892.491,E2 -15892.491} C_VEL
LIN {X 0,Y 336.648,Z 903.005,A -85,B 0,C 180,E1 -15892.836,E2 -15892.836} C_VEL
LIN {X 0,Y 335.174,Z 916.339,A -85,B 0,C 180,E1 -15893.35,E2 -15893.35} C_VEL
LIN {X 0,Y 333.394,Z 929.454,A -85,B 0,C 180,E1 -15894.014,E2 -15894.014} C_VEL
LIN {X 0,Y 331.695,Z 940.841,A -85,B 0,C 180,E1 -15894.735,E2 -15894.735} C_VEL
LIN {X 0,Y 329.227,Z 954.072,A -85,B 0,C 180,E1 -15895.736,E2 -15895.736} C_VEL
LIN {X 0,Y 326.888,Z 965.947,A -85,B 0,C 180,E1 -15896.828,E2 -15896.828} C_VEL
LIN {X 0,Y 324.271,Z 977.824,A -85,B 0,C 180,E1 -15898.114,E2 -15898.114} C_VEL
LIN {X 0,Y 321.619,Z 988.602,A -85,B 0,C 180,E1 -15899.466,E2 -15899.466} C_VEL
LIN {X 0,Y 319.027,Z 999.101,A -85,B 0,C 180,E1 -15901.011,E2 -15901.011} C_VEL
LIN {X 0,Y 316.411,Z 1008.952,A -85,B 0,C 180,E1 -15902.681,E2 -15902.681} C_VEL
LIN {X 0,Y 313.988,Z 1018.103,A -85,B 0,C 180,E1 -15904.478,E2 -15904.478} C_VEL
LIN {X 0,Y 311.737,Z 1026.629,A -85,B 0,C 180,E1 -15906.412,E2 -15906.412} C_VEL
LIN {X 0,Y 309.485,Z 1035.231,A -85,B 0,C 180,E1 -15908.695,E2 -15908.695} C_VEL
LIN {X 0,Y 307.928,Z 1041.665,A -85,B 0,C 180,E1 -15910.675,E2 -15910.675} C_VEL
LIN {X 0,Y 306.18,Z 1048.927,A -85,B 0,C 180,E1 -15913.327,E2 -15913.327} C_VEL
LIN {X 0,Y 305.255,Z 1053.582,A -85,B 0,C 180,E1 -15915.33,E2 -15915.33} C_VEL
LIN {X 0,Y 304.384,Z 1058.683,A -85,B 0,C 180,E1 -15918.007,E2 -15918.007} C_VEL
LIN {X 0,Y 303.857,Z 1062.685,A -85,B 0,C 180,E1 -15920.683,E2 -15920.683} C_VEL
LIN {X 0,Y 303.679,Z 1065.645,A -85,B 0,C 180,E1 -15923.355,E2 -15923.355} C_VEL
LIN {X 0,Y 303.597,Z 1066.831,A -85,B 0,C 180,E1 -15924.687,E2 -15924.687} C_VEL
LIN {X 0,Y 303.588,Z 1068.302,A -85,B 0,C 180,E1 -15927.346,E2 -15927.346} C_VEL
LIN {X 0,Y 303.602,Z 1068.789,A -85,B 0,C 180,E1 -15930,E2 -15930} C_VEL
LIN {X 0,Y 303.588,Z 1068.302,A -85,B 0,C 180,E1 -15932.654,E2 -15932.654} C_VEL
LIN {X 0,Y 303.624,Z 1066.625,A -85,B 0,C 180,E1 -15935.544,E2 -15935.544} C_VEL
LIN {X 0,Y 303.697,Z 1064.36,A -85,B 0,C 180,E1 -15937.981,E2 -15937.981} C_VEL
LIN {X 0,Y 304.197,Z 1059.771,A -85,B 0,C 180,E1 -15941.325,E2 -15941.325} C_VEL
LIN {X 0,Y 304.777,Z 1056.281,A -85,B 0,C 180,E1 -15943.332,E2 -15943.332} C_VEL
LIN {X 0,Y 305.839,Z 1050.55,A -85,B 0,C 180,E1 -15946.006,E2 -15946.006} C_VEL
LIN {X 0,Y 306.97,Z 1045.488,A -85,B 0,C 180,E1 -15948.003,E2 -15948.003} C_VEL
LIN {X 0,Y 308.92,Z 1037.454,A -85,B 0,C 180,E1 -15950.648,E2 -15950.648} C_VEL
LIN {X 0,Y 310.675,Z 1030.468,A -85,B 0,C 180,E1 -15952.616,E2 -15952.616} C_VEL
LIN {X 0,Y 312.834,Z 1022.5,A -85,B 0,C 180,E1 -15954.557,E2 -15954.557} C_VEL
LIN {X 0,Y 315.315,Z 1013.389,A -85,B 0,C 180,E1 -15956.472,E2 -15956.472} C_VEL
LIN {X 0,Y 317.533,Z 1004.819,A -85,B 0,C 180,E1 -15958.055,E2 -15958.055} C_VEL
LIN {X 0,Y 320.345,Z 994.044,A -85,B 0,C 180,E1 -15959.759,E2 -15959.759} C_VEL
LIN {X 0,Y 323.031,Z 982.79,A -85,B 0,C 180,E1 -15961.293,E2 -15961.293} C_VEL
LIN {X 0,Y 325.727,Z 971.123,A -85,B 0,C 180,E1 -15962.642,E2 -15962.642} C_VEL
LIN {X 0,Y 328.287,Z 959.1,A -85,B 0,C 180,E1 -15963.821,E2 -15963.821} C_VEL
LIN {X 0,Y 330.62,Z 946.782,A -85,B 0,C 180,E1 -15964.839,E2 -15964.839} C_VEL
LIN {X 0,Y 332.713,Z 934.24,A -85,B 0,C 180,E1 -15965.698,E2 -15965.698} C_VEL
LIN {X 0,Y 334.542,Z 920.812,A -85,B 0,C 180,E1 -15966.449,E2 -15966.449} C_VEL
LIN {X 0,Y 336.136,Z 907.899,A -85,B 0,C 180,E1 -15966.995,E2 -15966.995} C_VEL
LIN {X 0,Y 337.393,Z 894.424,A -85,B 0,C 180,E1 -15967.417,E2 -15967.417} C_VEL
LIN {X 0,Y 338.653,Z 864.211,A -85,B 0,C 180,E1 -15968.11,E2 -15968.11} C_VEL
LIN {X 0,Y 343.173,Z 754.794,A -85,B 0,C 180,E1 -15970.402,E2 -15970.402} C_VEL
LIN {X 0,Y 342.767,Z 751.671,A -85,B 0,C 180,E1 -15970.543,E2 -15970.543} C_VEL
LIN {X 0,Y 336.3,Z 737.35,A -85,B 0,C 180,E1 -15971.885,E2 -15971.885} C_VEL
LIN {X 0,Y 327.689,Z 720.455,A -85,B 0,C 180,E1 -15973.739,E2 -15973.739} C_VEL
LIN {X 0,Y 319.633,Z 706.288,A -85,B 0,C 180,E1 -15975.569,E2 -15975.569} C_VEL
LIN {X 0,Y 313.541,Z 696.292,A -85,B 0,C 180,E1 -15977.035,E2 -15977.035} C_VEL
LIN {X 0,Y 309.945,Z 690.728,A -85,B 0,C 180,E1 -15977.936,E2 -15977.936} C_VEL
LIN {X 0,Y 307.527,Z 686.622,A -85,B 0,C 180,E1 -15978.641,E2 -15978.641} C_VEL
LIN {X 0,Y 305.542,Z 680.532,A -85,B 0,C 180,E1 -15981.162,E2 -15981.162} C_VEL
LIN {X 0,Y 305.516,Z 680.237,A -85,B 0,C 180,E1 -15981.603,E2 -15981.603} C_VEL
LIN {X 0,Y 305.457,Z 680.207,A -85,B 0,C 180,E1 -15984.886,E2 -15984.886} C_VEL
LIN {X 0,Y 305.446,Z 680.229,A -85,B 0,C 180,E1 -15988.354,E2 -15988.354} C_VEL
LIN {X 0,Y 305.514,Z 680.173,A -85,B 0,C 180,E1 -15991.113,E2 -15991.113} C_VEL
LIN {X 0,Y 305.565,Z 680.214,A -85,B 0,C 180,E1 -15994.087,E2 -15994.087} C_VEL
LIN {X 0,Y 305.497,Z 680.229,A -85,B 0,C 180,E1 -15998.402,E2 -15998.402} C_VEL
LIN {X 0,Y 305.585,Z 680.218,A -85,B 0,C 180,E1 -16001.217,E2 -16001.217} C_VEL
LIN {X 0,Y 305.642,Z 680.221,A -85,B 0,C 180,E1 -16005.348,E2 -16005.348} C_VEL
LIN {X 0,Y 305.633,Z 680.226,A -85,B 0,C 180,E1 -16009.399,E2 -16009.399} C_VEL
LIN {X 0,Y 305.802,Z 680.18,A -85,B 0,C 180,E1 -16012.074,E2 -16012.074} C_VEL
LIN {X 0,Y 305.684,Z 680.218,A -85,B 0,C 180,E1 -16014.723,E2 -16014.723} C_VEL
LIN {X 0,Y 305.951,Z 680.176,A -85,B 0,C 180,E1 -16018.683,E2 -16018.683} C_VEL
LIN {X 0,Y 305.951,Z 680.17,A -85,B 0,C 180,E1 -16021.316,E2 -16021.316} C_VEL
LIN {X 0,Y 305.84,Z 680.187,A -85,B 0,C 180,E1 -16026.597,E2 -16026.597} C_VEL
LIN {X 0,Y 305.728,Z 680.206,A -85,B 0,C 180,E1 -16029.26,E2 -16029.26} C_VEL
LIN {X 0,Y 305.579,Z 680.211,A -85,B 0,C 180,E1 -16033.296,E2 -16033.296} C_VEL
LIN {X 0,Y 305.585,Z 680.226,A -85,B 0,C 180,E1 -16036.02,E2 -16036.02} C_VEL
LIN {X 0,Y 305.596,Z 680.228,A -85,B 0,C 180,E1 -16039.459,E2 -16039.459} C_VEL
LIN {X 0,Y 305.501,Z 680.228,A -85,B 0,C 180,E1 -16043.049,E2 -16043.049} C_VEL
LIN {X 0,Y 305.525,Z 680.208,A -85,B 0,C 180,E1 -16046.221,E2 -16046.221} C_VEL
LIN {X 0,Y 305.487,Z 680.178,A -85,B 0,C 180,E1 -16049.05,E2 -16049.05} C_VEL
LIN {X 0,Y 305.437,Z 680.243,A -85,B 0,C 180,E1 -16051.952,E2 -16051.952} C_VEL
LIN {X 0,Y 305.455,Z 680.199,A -85,B 0,C 180,E1 -16055.113,E2 -16055.113} C_VEL
LIN {X 0,Y 305.477,Z 680.223,A -85,B 0,C 180,E1 -16058.537,E2 -16058.537} C_VEL
LIN {X 0,Y 305.496,Z 680.386,A -85,B 0,C 180,E1 -16060.998,E2 -16060.998} C_VEL
LIN {X 0,Y 305.787,Z 681.644,A -85,B 0,C 180,E1 -16061.415,E2 -16061.415} C_VEL
LIN {X 0,Y 307.145,Z 683.96,A -85,B 0,C 180,E1 -16061.89,E2 -16061.89} C_VEL
LIN {X 0,Y 309.608,Z 686.139,A -85,B 0,C 180,E1 -16062.629,E2 -16062.629} C_VEL
LIN {X 0,Y 311.862,Z 689.458,A -85,B 0,C 180,E1 -16063.349,E2 -16063.349} C_VEL
LIN {X 0,Y 314.464,Z 691.814,A -85,B 0,C 180,E1 -16064.206,E2 -16064.206} C_VEL
LIN {X 0,Y 316.953,Z 695.131,A -85,B 0,C 180,E1 -16065.048,E2 -16065.048} C_VEL
LIN {X 0,Y 319.928,Z 697.783,A -85,B 0,C 180,E1 -16066.102,E2 -16066.102} C_VEL
LIN {X 0,Y 322.565,Z 701.151,A -85,B 0,C 180,E1 -16067.073,E2 -16067.073} C_VEL
LIN {X 0,Y 325.397,Z 703.659,A -85,B 0,C 180,E1 -16068.139,E2 -16068.139} C_VEL
LIN {X 0,Y 328.312,Z 707.265,A -85,B 0,C 180,E1 -16069.304,E2 -16069.304} C_VEL
LIN {X 0,Y 330.924,Z 709.542,A -85,B 0,C 180,E1 -16070.312,E2 -16070.312} C_VEL
LIN {X 0,Y 333.948,Z 713.113,A -85,B 0,C 180,E1 -16071.544,E2 -16071.544} C_VEL
LIN {X 0,Y 336.591,Z 715.424,A -85,B 0,C 180,E1 -16072.605,E2 -16072.605} C_VEL
LIN {X 0,Y 339.976,Z 719.287,A -85,B 0,C 180,E1 -16074.041,E2 -16074.041} C_VEL
LIN {X 0,Y 342.642,Z 721.591,A -85,B 0,C 180,E1 -16075.173,E2 -16075.173} C_VEL
LIN {X 0,Y 346.218,Z 725.542,A -85,B 0,C 180,E1 -16076.765,E2 -16076.765} C_VEL
LIN {X 0,Y 349.261,Z 728.068,A -85,B 0,C 180,E1 -16078.128,E2 -16078.128} C_VEL
LIN {X 0,Y 352.877,Z 731.979,A -85,B 0,C 180,E1 -16079.859,E2 -16079.859} C_VEL
LIN {X 0,Y 355.755,Z 734.255,A -85,B 0,C 180,E1 -16081.248,E2 -16081.248} C_VEL
LIN {X 0,Y 358.617,Z 737.578,A -85,B 0,C 180,E1 -16082.754,E2 -16082.754} C_VEL
LIN {X 0,Y 361.892,Z 740.046,A -85,B 0,C 180,E1 -16084.484,E2 -16084.484} C_VEL
LIN {X 0,Y 365.581,Z 744.188,A -85,B 0,C 180,E1 -16086.643,E2 -16086.643} C_VEL
LIN {X 0,Y 368.761,Z 746.481,A -85,B 0,C 180,E1 -16088.581,E2 -16088.581} C_VEL
LIN {X 0,Y 369.914,Z 747.353,A -85,B 0,C 180,E1 -16089.313,E2 -16089.313} C_VEL
LIN {X 0,Y 372.315,Z 750.229,A -85,B 0,C 180,E1 -16091.039,E2 -16091.039} C_VEL
LIN {X 0,Y 375.037,Z 752.478,A -85,B 0,C 180,E1 -16093.072,E2 -16093.072} C_VEL
LIN {X 0,Y 377.542,Z 753.95,A -85,B 0,C 180,E1 -16095.136,E2 -16095.136} C_VEL
LIN {X 0,Y 379.355,Z 756.418,A -85,B 0,C 180,E1 -16096.95,E2 -16096.95} C_VEL
LIN {X 0,Y 381.186,Z 758.22,A -85,B 0,C 180,E1 -16099.046,E2 -16099.046} C_VEL
LIN {X 0,Y 383.094,Z 759.342,A -85,B 0,C 180,E1 -16101.561,E2 -16101.561} C_VEL
LIN {X 0,Y 384.545,Z 760.063,A -85,B 0,C 180,E1 -16104.16,E2 -16104.16} C_VEL
LIN {X 0,Y 385.204,Z 760.511,A -85,B 0,C 180,E1 -16105.815,E2 -16105.815} C_VEL
LIN {X 0,Y 385.734,Z 760.711,A -85,B 0,C 180,E1 -16107.912,E2 -16107.912} C_VEL
LIN {X 0,Y 385.935,Z 760.774,A -85,B 0,C 180,E1 -16110,E2 -16110} C_VEL
LIN {X 0,Y 385.734,Z 760.712,A -85,B 0,C 180,E1 -16112.088,E2 -16112.088} C_VEL
LIN {X 0,Y 385.051,Z 760.372,A -85,B 0,C 180,E1 -16114.625,E2 -16114.625} C_VEL
LIN {X 0,Y 383.771,Z 759.634,A -85,B 0,C 180,E1 -16117.365,E2 -16117.365} C_VEL
LIN {X 0,Y 381.926,Z 758.745,A -85,B 0,C 180,E1 -16120.058,E2 -16120.058} C_VEL
LIN {X 0,Y 379.871,Z 757.006,A -85,B 0,C 180,E1 -16122.459,E2 -16122.459} C_VEL
LIN {X 0,Y 377.894,Z 754.518,A -85,B 0,C 180,E1 -16124.529,E2 -16124.529} C_VEL
LIN {X 0,Y 377.051,Z 753.512,A -85,B 0,C 180,E1 -16125.31,E2 -16125.31} C_VEL
LIN {X 0,Y 374.307,Z 751.938,A -85,B 0,C 180,E1 -16127.482,E2 -16127.482} C_VEL
LIN {X 0,Y 371.537,Z 749.415,A -85,B 0,C 180,E1 -16129.545,E2 -16129.545} C_VEL
LIN {X 0,Y 369.539,Z 746.905,A -85,B 0,C 180,E1 -16130.954,E2 -16130.954} C_VEL
LIN {X 0,Y 365.956,Z 744.493,A -85,B 0,C 180,E1 -16133.129,E2 -16133.129} C_VEL
LIN {X 0,Y 362.863,Z 741.157,A -85,B 0,C 180,E1 -16134.977,E2 -16134.977} C_VEL
LIN {X 0,Y 361.893,Z 740.041,A -85,B 0,C 180,E1 -16135.516,E2 -16135.516} C_VEL
LIN {X 0,Y 358.66,Z 737.612,A -85,B 0,C 180,E1 -16137.224,E2 -16137.224} C_VEL
LIN {X 0,Y 355.625,Z 734.112,A -85,B 0,C 180,E1 -16138.82,E2 -16138.82} C_VEL
LIN {X 0,Y 351.423,Z 730.585,A -85,B 0,C 180,E1 -16140.827,E2 -16140.827} C_VEL
LIN {X 0,Y 348.309,Z 727.116,A -85,B 0,C 180,E1 -16142.301,E2 -16142.301} C_VEL
LIN {X 0,Y 344.954,Z 724.325,A -85,B 0,C 180,E1 -16143.787,E2 -16143.787} C_VEL
LIN {X 0,Y 341.674,Z 720.638,A -85,B 0,C 180,E1 -16145.241,E2 -16145.241} C_VEL
LIN {X 0,Y 338.356,Z 717.659,A -85,B 0,C 180,E1 -16146.631,E2 -16146.631} C_VEL
LIN {X 0,Y 336.002,Z 714.752,A -85,B 0,C 180,E1 -16147.636,E2 -16147.636} C_VEL
LIN {X 0,Y 332.561,Z 711.686,A -85,B 0,C 180,E1 -16149.013,E2 -16149.013} C_VEL
LIN {X 0,Y 330.2,Z 708.774,A -85,B 0,C 180,E1 -16149.985,E2 -16149.985} C_VEL
LIN {X 0,Y 326.87,Z 705.697,A -85,B 0,C 180,E1 -16151.268,E2 -16151.268} C_VEL
LIN {X 0,Y 324.622,Z 702.864,A -85,B 0,C 180,E1 -16152.154,E2 -16152.154} C_VEL
LIN {X 0,Y 321.498,Z 700.001,A -85,B 0,C 180,E1 -16153.311,E2 -16153.311} C_VEL
LIN {X 0,Y 319.464,Z 697.214,A -85,B 0,C 180,E1 -16154.069,E2 -16154.069} C_VEL
LIN {X 0,Y 316.661,Z 694.83,A -85,B 0,C 180,E1 -16155.049,E2 -16155.049} C_VEL
LIN {X 0,Y 313.767,Z 691.113,A -85,B 0,C 180,E1 -16156.024,E2 -16156.024} C_VEL
LIN {X 0,Y 311.122,Z 688.578,A -85,B 0,C 180,E1 -16156.886,E2 -16156.886} C_VEL
LIN {X 0,Y 309.285,Z 685.687,A -85,B 0,C 180,E1 -16157.473,E2 -16157.473} C_VEL
LIN {X 0,Y 306.815,Z 683.593,A -85,B 0,C 180,E1 -16158.214,E2 -16158.214} C_VEL
LIN {X 0,Y 305.592,Z 680.909,A -85,B 0,C 180,E1 -16158.764,E2 -16158.764} C_VEL
LIN {X 0,Y 305.488,Z 680.288,A -85,B 0,C 180,E1 -16159.169,E2 -16159.169} C_VEL
LIN {X 0,Y 305.503,Z 680.216,A -85,B 0,C 180,E1 -16161.602,E2 -16161.602} C_VEL
LIN {X 0,Y 305.455,Z 680.199,A -85,B 0,C 180,E1 -16164.887,E2 -16164.887} C_VEL
LIN {X 0,Y 305.444,Z 680.232,A -85,B 0,C 180,E1 -16168.355,E2 -16168.355} C_VEL
LIN {X 0,Y 305.512,Z 680.174,A -85,B 0,C 180,E1 -16171.114,E2 -16171.114} C_VEL
LIN {X 0,Y 305.565,Z 680.213,A -85,B 0,C 180,E1 -16174.088,E2 -16174.088} C_VEL
LIN {X 0,Y 305.501,Z 680.228,A -85,B 0,C 180,E1 -16178.403,E2 -16178.403} C_VEL
LIN {X 0,Y 305.585,Z 680.219,A -85,B 0,C 180,E1 -16181.218,E2 -16181.218} C_VEL
LIN {X 0,Y 305.641,Z 680.22,A -85,B 0,C 180,E1 -16185.349,E2 -16185.349} C_VEL
LIN {X 0,Y 305.63,Z 680.223,A -85,B 0,C 180,E1 -16189.4,E2 -16189.4} C_VEL
LIN {X 0,Y 305.796,Z 680.183,A -85,B 0,C 180,E1 -16192.074,E2 -16192.074} C_VEL
LIN {X 0,Y 305.683,Z 680.221,A -85,B 0,C 180,E1 -16194.724,E2 -16194.724} C_VEL
LIN {X 0,Y 305.951,Z 680.172,A -85,B 0,C 180,E1 -16198.684,E2 -16198.684} C_VEL
LIN {X 0,Y 305.951,Z 680.177,A -85,B 0,C 180,E1 -16201.317,E2 -16201.317} C_VEL
LIN {X 0,Y 305.89,Z 680.175,A -85,B 0,C 180,E1 -16202.071,E2 -16202.071} C_VEL
LIN {X 0,Y 305.184,Z 680.265,A -85,B 0,C 180,E1 -16203.168,E2 -16203.168} C_VEL
LIN {X 0,Y 302.283,Z 680.641,A -85,B 0,C 180,E1 -16204.953,E2 -16204.953} C_VEL
LIN {X 0,Y 299.85,Z 680.935,A -85,B 0,C 180,E1 -16206.401,E2 -16206.401} C_VEL
LIN {X 0,Y 298.82,Z 681.05,A -85,B 0,C 180,E1 -16207.524,E2 -16207.524} C_VEL
LIN {X 0,Y 298.743,Z 681.058,A -85,B 0,C 180,E1 -16207.904,E2 -16207.904} C_VEL
LIN {X 0,Y 298.588,Z 681.1,A -85,B 0,C 180,E1 -16210.854,E2 -16210.854} C_VEL
LIN {X 0,Y 298.578,Z 681.103,A -85,B 0,C 180,E1 -16215.195,E2 -16215.195} C_VEL
LIN {X 0,Y 298.536,Z 681.101,A -85,B 0,C 180,E1 -16219.244,E2 -16219.244} C_VEL
LIN {X 0,Y 298.451,Z 681.109,A -85,B 0,C 180,E1 -16223.598,E2 -16223.598} C_VEL
LIN {X 0,Y 298.481,Z 681.075,A -85,B 0,C 180,E1 -16226.575,E2 -16226.575} C_VEL
LIN {X 0,Y 298.415,Z 681.06,A -85,B 0,C 180,E1 -16229.642,E2 -16229.642} C_VEL
LIN {X 0,Y 298.39,Z 681.13,A -85,B 0,C 180,E1 -16232.801,E2 -16232.801} C_VEL
LIN {X 0,Y 298.466,Z 681.081,A -85,B 0,C 180,E1 -16236.815,E2 -16236.815} C_VEL
LIN {X 0,Y 298.506,Z 681.427,A -85,B 0,C 180,E1 -16237.612,E2 -16237.612} C_VEL
LIN {X 0,Y 300.156,Z 686.383,A -85,B 0,C 180,E1 -16239.754,E2 -16239.754} C_VEL
LIN {X 0,Y 303.053,Z 691.033,A -85,B 0,C 180,E1 -16240.621,E2 -16240.621} C_VEL
LIN {X 0,Y 308.274,Z 699.097,A -85,B 0,C 180,E1 -16242.007,E2 -16242.007} C_VEL
LIN {X 0,Y 311.739,Z 704.652,A -85,B 0,C 180,E1 -16242.888,E2 -16242.888} C_VEL
LIN {X 0,Y 319.431,Z 717.759,A -85,B 0,C 180,E1 -16244.753,E2 -16244.753} C_VEL
LIN {X 0,Y 326.475,Z 731.03,A -85,B 0,C 180,E1 -16246.373,E2 -16246.373} C_VEL
LIN {X 0,Y 334.343,Z 747.252,A -85,B 0,C 180,E1 -16248.095,E2 -16248.095} C_VEL
LIN {X 0,Y 337.74,Z 755.016,A -85,B 0,C 180,E1 -16248.821,E2 -16248.821} C_VEL
LIN {X 0,Y 331.914,Z 891.127,A -85,B 0,C 180,E1 -16251.749,E2 -16251.749} C_VEL
LIN {X 0,Y 331.015,Z 902.799,A -85,B 0,C 180,E1 -16252.093,E2 -16252.093} C_VEL
LIN {X 0,Y 329.497,Z 916.133,A -85,B 0,C 180,E1 -16252.612,E2 -16252.612} C_VEL
LIN {X 0,Y 327.668,Z 929.248,A -85,B 0,C 180,E1 -16253.283,E2 -16253.283} C_VEL
LIN {X 0,Y 325.885,Z 940.634,A -85,B 0,C 180,E1 -16254.009,E2 -16254.009} C_VEL
LIN {X 0,Y 323.363,Z 953.866,A -85,B 0,C 180,E1 -16255.025,E2 -16255.025} C_VEL
LIN {X 0,Y 320.92,Z 965.74,A -85,B 0,C 180,E1 -16256.129,E2 -16256.129} C_VEL
LIN {X 0,Y 318.133,Z 977.958,A -85,B 0,C 180,E1 -16257.475,E2 -16257.475} C_VEL
LIN {X 0,Y 315.451,Z 988.394,A -85,B 0,C 180,E1 -16258.803,E2 -16258.803} C_VEL
LIN {X 0,Y 312.742,Z 998.893,A -85,B 0,C 180,E1 -16260.371,E2 -16260.371} C_VEL
LIN {X 0,Y 309.822,Z 1009.48,A -85,B 0,C 180,E1 -16262.212,E2 -16262.212} C_VEL
LIN {X 0,Y 307.06,Z 1019.359,A -85,B 0,C 180,E1 -16264.224,E2 -16264.224} C_VEL
LIN {X 0,Y 304.77,Z 1027.7,A -85,B 0,C 180,E1 -16266.2,E2 -16266.2} C_VEL
LIN {X 0,Y 302.793,Z 1035.023,A -85,B 0,C 180,E1 -16268.201,E2 -16268.201} C_VEL
LIN {X 0,Y 301.139,Z 1041.457,A -85,B 0,C 180,E1 -16270.221,E2 -16270.221} C_VEL
LIN {X 0,Y 299.286,Z 1048.719,A -85,B 0,C 180,E1 -16272.931,E2 -16272.931} C_VEL
LIN {X 0,Y 298.292,Z 1053.442,A -85,B 0,C 180,E1 -16275.015,E2 -16275.015} C_VEL
LIN {X 0,Y 297.367,Z 1058.475,A -85,B 0,C 180,E1 -16277.719,E2 -16277.719} C_VEL
LIN {X 0,Y 296.775,Z 1062.477,A -85,B 0,C 180,E1 -16280.458,E2 -16280.458} C_VEL
LIN {X 0,Y 296.575,Z 1065.438,A -85,B 0,C 180,E1 -16283.195,E2 -16283.195} C_VEL
LIN {X 0,Y 296.511,Z 1066.625,A -85,B 0,C 180,E1 -16284.56,E2 -16284.56} C_VEL
LIN {X 0,Y 296.513,Z 1068.097,A -85,B 0,C 180,E1 -16287.283,E2 -16287.283} C_VEL
LIN {X 0,Y 296.517,Z 1068.584,A -85,B 0,C 180,E1 -16290,E2 -16290} C_VEL
LIN {X 0,Y 296.513,Z 1068.097,A -85,B 0,C 180,E1 -16292.717,E2 -16292.717} C_VEL
LIN {X 0,Y 296.511,Z 1066.625,A -85,B 0,C 180,E1 -16295.44,E2 -16295.44} C_VEL
LIN {X 0,Y 296.63,Z 1064.153,A -85,B 0,C 180,E1 -16298.172,E2 -16298.172} C_VEL
LIN {X 0,Y 297.165,Z 1059.564,A -85,B 0,C 180,E1 -16301.597,E2 -16301.597} C_VEL
LIN {X 0,Y 297.797,Z 1056.073,A -85,B 0,C 180,E1 -16303.65,E2 -16303.65} C_VEL
LIN {X 0,Y 298.915,Z 1050.341,A -85,B 0,C 180,E1 -16306.388,E2 -16306.388} C_VEL
LIN {X 0,Y 300.116,Z 1045.279,A -85,B 0,C 180,E1 -16308.429,E2 -16308.429} C_VEL
LIN {X 0,Y 302.194,Z 1037.246,A -85,B 0,C 180,E1 -16311.129,E2 -16311.129} C_VEL
LIN {X 0,Y 304.039,Z 1030.259,A -85,B 0,C 180,E1 -16313.138,E2 -16313.138} C_VEL
LIN {X 0,Y 306.294,Z 1022.292,A -85,B 0,C 180,E1 -16315.118,E2 -16315.118} C_VEL
LIN {X 0,Y 308.878,Z 1013.18,A -85,B 0,C 180,E1 -16317.068,E2 -16317.068} C_VEL
LIN {X 0,Y 311.192,Z 1004.61,A -85,B 0,C 180,E1 -16318.679,E2 -16318.679} C_VEL
LIN {X 0,Y 314.314,Z 992.745,A -85,B 0,C 180,E1 -16320.575,E2 -16320.575} C_VEL
LIN {X 0,Y 316.918,Z 982.582,A -85,B 0,C 180,E1 -16321.968,E2 -16321.968} C_VEL
LIN {X 0,Y 319.87,Z 970.335,A -85,B 0,C 180,E1 -16323.393,E2 -16323.393} C_VEL
LIN {X 0,Y 322.367,Z 958.893,A -85,B 0,C 180,E1 -16324.529,E2 -16324.529} C_VEL
LIN {X 0,Y 324.791,Z 946.576,A -85,B 0,C 180,E1 -16325.557,E2 -16325.557} C_VEL
LIN {X 0,Y 326.922,Z 934.033,A -85,B 0,C 180,E1 -16326.431,E2 -16326.431} C_VEL
LIN {X 0,Y 328.862,Z 920.607,A -85,B 0,C 180,E1 -16327.184,E2 -16327.184} C_VEL
LIN {X 0,Y 330.493,Z 907.694,A -85,B 0,C 180,E1 -16327.736,E2 -16327.736} C_VEL
LIN {X 0,Y 331.723,Z 895,A -85,B 0,C 180,E1 -16328.144,E2 -16328.144} C_VEL
LIN {X 0,Y 332.884,Z 868.739,A -85,B 0,C 180,E1 -16328.765,E2 -16328.765} C_VEL
LIN {X 0,Y 337.734,Z 756.068,A -85,B 0,C 180,E1 -16331.151,E2 -16331.151} C_VEL
LIN {X 0,Y 337.401,Z 754.214,A -85,B 0,C 180,E1 -16331.251,E2 -16331.251} C_VEL
LIN {X 0,Y 331.486,Z 741.127,A -85,B 0,C 180,E1 -16332.522,E2 -16332.522} C_VEL
LIN {X 0,Y 323.348,Z 724.925,A -85,B 0,C 180,E1 -16334.338,E2 -16334.338} C_VEL
LIN {X 0,Y 315.43,Z 710.858,A -85,B 0,C 180,E1 -16336.201,E2 -16336.201} C_VEL
LIN {X 0,Y 309.637,Z 701.206,A -85,B 0,C 180,E1 -16337.645,E2 -16337.645} C_VEL
LIN {X 0,Y 303.202,Z 691.22,A -85,B 0,C 180,E1 -16339.34,E2 -16339.34} C_VEL
LIN {X 0,Y 300.077,Z 686.235,A -85,B 0,C 180,E1 -16340.288,E2 -16340.288} C_VEL
LIN {X 0,Y 298.454,Z 681.256,A -85,B 0,C 180,E1 -16342.513,E2 -16342.513} C_VEL
LIN {X 0,Y 298.402,Z 681.093,A -85,B 0,C 180,E1 -16345.58,E2 -16345.58} C_VEL
LIN {X 0,Y 298.389,Z 681.092,A -85,B 0,C 180,E1 -16348.79,E2 -16348.79} C_VEL
LIN {X 0,Y 298.457,Z 681.053,A -85,B 0,C 180,E1 -16351.903,E2 -16351.903} C_VEL
LIN {X 0,Y 298.48,Z 681.116,A -85,B 0,C 180,E1 -16354.923,E2 -16354.923} C_VEL
LIN {X 0,Y 298.45,Z 681.12,A -85,B 0,C 180,E1 -16359.315,E2 -16359.315} C_VEL
LIN {X 0,Y 298.531,Z 681.091,A -85,B 0,C 180,E1 -16362.179,E2 -16362.179} C_VEL
LIN {X 0,Y 298.586,Z 681.102,A -85,B 0,C 180,E1 -16364.994,E2 -16364.994} C_VEL
LIN {X 0,Y 298.588,Z 681.102,A -85,B 0,C 180,E1 -16369.146,E2 -16369.146} C_VEL
LIN {X 0,Y 298.748,Z 681.058,A -85,B 0,C 180,E1 -16371.885,E2 -16371.885} C_VEL
LIN {X 0,Y 298.654,Z 681.093,A -85,B 0,C 180,E1 -16374.598,E2 -16374.598} C_VEL
LIN {X 0,Y 298.917,Z 681.05,A -85,B 0,C 180,E1 -16378.652,E2 -16378.652} C_VEL
LIN {X 0,Y 298.917,Z 681.045,A -85,B 0,C 180,E1 -16381.347,E2 -16381.347} C_VEL
LIN {X 0,Y 298.786,Z 681.063,A -85,B 0,C 180,E1 -16386.754,E2 -16386.754} C_VEL
LIN {X 0,Y 298.673,Z 681.087,A -85,B 0,C 180,E1 -16389.48,E2 -16389.48} C_VEL
LIN {X 0,Y 298.543,Z 681.089,A -85,B 0,C 180,E1 -16393.615,E2 -16393.615} C_VEL
LIN {X 0,Y 298.54,Z 681.098,A -85,B 0,C 180,E1 -16396.409,E2 -16396.409} C_VEL
LIN {X 0,Y 298.526,Z 681.11,A -85,B 0,C 180,E1 -16399.666,E2 -16399.666} C_VEL
LIN {X 0,Y 298.458,Z 681.111,A -85,B 0,C 180,E1 -16403.597,E2 -16403.597} C_VEL
LIN {X 0,Y 298.48,Z 681.074,A -85,B 0,C 180,E1 -16406.575,E2 -16406.575} C_VEL
LIN {X 0,Y 298.413,Z 681.062,A -85,B 0,C 180,E1 -16409.641,E2 -16409.641} C_VEL
LIN {X 0,Y 298.388,Z 681.13,A -85,B 0,C 180,E1 -16412.8,E2 -16412.8} C_VEL
LIN {X 0,Y 298.445,Z 681.067,A -85,B 0,C 180,E1 -16416.809,E2 -16416.809} C_VEL
LIN {X 0,Y 298.442,Z 681.317,A -85,B 0,C 180,E1 -16419.33,E2 -16419.33} C_VEL
LIN {X 0,Y 298.652,Z 682.213,A -85,B 0,C 180,E1 -16419.666,E2 -16419.666} C_VEL
LIN {X 0,Y 300.077,Z 684.858,A -85,B 0,C 180,E1 -16420.174,E2 -16420.174} C_VEL
LIN {X 0,Y 302.253,Z 686.864,A -85,B 0,C 180,E1 -16420.78,E2 -16420.78} C_VEL
LIN {X 0,Y 304.39,Z 689.962,A -85,B 0,C 180,E1 -16421.405,E2 -16421.405} C_VEL
LIN {X 0,Y 306.946,Z 692.475,A -85,B 0,C 180,E1 -16422.181,E2 -16422.181} C_VEL
LIN {X 0,Y 309.527,Z 695.893,A -85,B 0,C 180,E1 -16422.991,E2 -16422.991} C_VEL
LIN {X 0,Y 312.18,Z 698.391,A -85,B 0,C 180,E1 -16423.822,E2 -16423.822} C_VEL
LIN {X 0,Y 314.958,Z 701.756,A -85,B 0,C 180,E1 -16424.761,E2 -16424.761} C_VEL
LIN {X 0,Y 317.726,Z 704.228,A -85,B 0,C 180,E1 -16425.689,E2 -16425.689} C_VEL
LIN {X 0,Y 320.753,Z 707.866,A -85,B 0,C 180,E1 -16426.801,E2 -16426.801} C_VEL
LIN {X 0,Y 323.346,Z 710.169,A -85,B 0,C 180,E1 -16427.758,E2 -16427.758} C_VEL
LIN {X 0,Y 326.524,Z 713.919,A -85,B 0,C 180,E1 -16429.004,E2 -16429.004} C_VEL
LIN {X 0,Y 329.111,Z 716.243,A -85,B 0,C 180,E1 -16429.992,E2 -16429.992} C_VEL
LIN {X 0,Y 332.514,Z 720.073,A -85,B 0,C 180,E1 -16431.368,E2 -16431.368} C_VEL
LIN {X 0,Y 334.905,Z 722.189,A -85,B 0,C 180,E1 -16432.335,E2 -16432.335} C_VEL
LIN {X 0,Y 338.199,Z 725.895,A -85,B 0,C 180,E1 -16433.721,E2 -16433.721} C_VEL
LIN {X 0,Y 341.003,Z 728.353,A -85,B 0,C 180,E1 -16434.897,E2 -16434.897} C_VEL
LIN {X 0,Y 344.603,Z 732.236,A -85,B 0,C 180,E1 -16436.487,E2 -16436.487} C_VEL
LIN {X 0,Y 347.855,Z 735.001,A -85,B 0,C 180,E1 -16437.936,E2 -16437.936} C_VEL
LIN {X 0,Y 351.562,Z 738.866,A -85,B 0,C 180,E1 -16439.678,E2 -16439.678} C_VEL
LIN {X 0,Y 354.353,Z 741.123,A -85,B 0,C 180,E1 -16441.018,E2 -16441.018} C_VEL
LIN {X 0,Y 357.382,Z 744.539,A -85,B 0,C 180,E1 -16442.596,E2 -16442.596} C_VEL
LIN {X 0,Y 361.163,Z 747.548,A -85,B 0,C 180,E1 -16444.601,E2 -16444.601} C_VEL
LIN {X 0,Y 364.439,Z 751.154,A -85,B 0,C 180,E1 -16446.502,E2 -16446.502} C_VEL
LIN {X 0,Y 367.688,Z 753.465,A -85,B 0,C 180,E1 -16448.475,E2 -16448.475} C_VEL
LIN {X 0,Y 368.67,Z 754.188,A -85,B 0,C 180,E1 -16449.08,E2 -16449.08} C_VEL
LIN {X 0,Y 371.248,Z 757.227,A -85,B 0,C 180,E1 -16450.918,E2 -16450.918} C_VEL
LIN {X 0,Y 374.09,Z 759.499,A -85,B 0,C 180,E1 -16453.028,E2 -16453.028} C_VEL
LIN {X 0,Y 376.479,Z 760.925,A -85,B 0,C 180,E1 -16454.98,E2 -16454.98} C_VEL
LIN {X 0,Y 378.539,Z 763.579,A -85,B 0,C 180,E1 -16457.024,E2 -16457.024} C_VEL
LIN {X 0,Y 380.288,Z 765.265,A -85,B 0,C 180,E1 -16459.019,E2 -16459.019} C_VEL
LIN {X 0,Y 382.213,Z 766.375,A -85,B 0,C 180,E1 -16461.541,E2 -16461.541} C_VEL
LIN {X 0,Y 383.671,Z 767.108,A -85,B 0,C 180,E1 -16464.147,E2 -16464.147} C_VEL
LIN {X 0,Y 384.333,Z 767.557,A -85,B 0,C 180,E1 -16465.805,E2 -16465.805} C_VEL
LIN {X 0,Y 384.87,Z 767.749,A -85,B 0,C 180,E1 -16467.907,E2 -16467.907} C_VEL
LIN {X 0,Y 385.07,Z 767.821,A -85,B 0,C 180,E1 -16470,E2 -16470} C_VEL
LIN {X 0,Y 384.87,Z 767.75,A -85,B 0,C 180,E1 -16472.093,E2 -16472.093} C_VEL
LIN {X 0,Y 384.181,Z 767.421,A -85,B 0,C 180,E1 -16474.636,E2 -16474.636} C_VEL
LIN {X 0,Y 382.892,Z 766.698,A -85,B 0,C 180,E1 -16477.382,E2 -16477.382} C_VEL
LIN {X 0,Y 381.038,Z 765.789,A -85,B 0,C 180,E1 -16480.082,E2 -16480.082} C_VEL
LIN {X 0,Y 378.963,Z 764.076,A -85,B 0,C 180,E1 -16482.489,E2 -16482.489} C_VEL
LIN {X 0,Y 376.882,Z 761.549,A -85,B 0,C 180,E1 -16484.633,E2 -16484.633} C_VEL
LIN {X 0,Y 376.126,Z 760.549,A -85,B 0,C 180,E1 -16485.349,E2 -16485.349} C_VEL
LIN {X 0,Y 373.251,Z 758.914,A -85,B 0,C 180,E1 -16487.607,E2 -16487.607} C_VEL
LIN {X 0,Y 370.314,Z 756.252,A -85,B 0,C 180,E1 -16489.755,E2 -16489.755} C_VEL
LIN {X 0,Y 368.109,Z 753.691,A -85,B 0,C 180,E1 -16491.269,E2 -16491.269} C_VEL
LIN {X 0,Y 364.44,Z 751.15,A -85,B 0,C 180,E1 -16493.498,E2 -16493.498} C_VEL
LIN {X 0,Y 361.057,Z 747.416,A -85,B 0,C 180,E1 -16495.46,E2 -16495.46} C_VEL
LIN {X 0,Y 356.807,Z 743.966,A -85,B 0,C 180,E1 -16497.707,E2 -16497.707} C_VEL
LIN {X 0,Y 353.412,Z 740.257,A -85,B 0,C 180,E1 -16499.432,E2 -16499.432} C_VEL
LIN {X 0,Y 349.712,Z 737.151,A -85,B 0,C 180,E1 -16501.183,E2 -16501.183} C_VEL
LIN {X 0,Y 346.629,Z 733.794,A -85,B 0,C 180,E1 -16502.626,E2 -16502.626} C_VEL
LIN {X 0,Y 342.913,Z 730.581,A -85,B 0,C 180,E1 -16504.269,E2 -16504.269} C_VEL
LIN {X 0,Y 339.878,Z 727.211,A -85,B 0,C 180,E1 -16505.595,E2 -16505.595} C_VEL
LIN {X 0,Y 336.421,Z 724.056,A -85,B 0,C 180,E1 -16507.032,E2 -16507.032} C_VEL
LIN {X 0,Y 333.894,Z 721.181,A -85,B 0,C 180,E1 -16508.077,E2 -16508.077} C_VEL
LIN {X 0,Y 330.394,Z 717.878,A -85,B 0,C 180,E1 -16509.473,E2 -16509.473} C_VEL
LIN {X 0,Y 328.113,Z 715.182,A -85,B 0,C 180,E1 -16510.394,E2 -16510.394} C_VEL
LIN {X 0,Y 324.691,Z 711.957,A -85,B 0,C 180,E1 -16511.715,E2 -16511.715} C_VEL
LIN {X 0,Y 322.528,Z 709.32,A -85,B 0,C 180,E1 -16512.559,E2 -16512.559} C_VEL
LIN {X 0,Y 319.174,Z 706.228,A -85,B 0,C 180,E1 -16513.758,E2 -16513.758} C_VEL
LIN {X 0,Y 316.879,Z 703.364,A -85,B 0,C 180,E1 -16514.615,E2 -16514.615} C_VEL
LIN {X 0,Y 313.37,Z 700.081,A -85,B 0,C 180,E1 -16515.761,E2 -16515.761} C_VEL
LIN {X 0,Y 311.328,Z 697.398,A -85,B 0,C 180,E1 -16516.467,E2 -16516.467} C_VEL
LIN {X 0,Y 308.288,Z 694.508,A -85,B 0,C 180,E1 -16517.383,E2 -16517.383} C_VEL
LIN {X 0,Y 306.3,Z 691.734,A -85,B 0,C 180,E1 -16518.021,E2 -16518.021} C_VEL
LIN {X 0,Y 303.602,Z 689.072,A -85,B 0,C 180,E1 -16518.816,E2 -16518.816} C_VEL
LIN {X 0,Y 301.904,Z 686.369,A -85,B 0,C 180,E1 -16519.323,E2 -16519.323} C_VEL
LIN {X 0,Y 299.666,Z 684.331,A -85,B 0,C 180,E1 -16519.949,E2 -16519.949} C_VEL
LIN {X 0,Y 298.55,Z 681.83,A -85,B 0,C 180,E1 -16520.428,E2 -16520.428} C_VEL
LIN {X 0,Y 298.432,Z 681.216,A -85,B 0,C 180,E1 -16520.818,E2 -16520.818} C_VEL
LIN {X 0,Y 298.413,Z 681.069,A -85,B 0,C 180,E1 -16523.93,E2 -16523.93} C_VEL
LIN {X 0,Y 298.388,Z 681.121,A -85,B 0,C 180,E1 -16527.983,E2 -16527.983} C_VEL
LIN {X 0,Y 298.455,Z 681.054,A -85,B 0,C 180,E1 -16531.904,E2 -16531.904} C_VEL
LIN {X 0,Y 298.481,Z 681.116,A -85,B 0,C 180,E1 -16534.924,E2 -16534.924} C_VEL
LIN {X 0,Y 298.453,Z 681.117,A -85,B 0,C 180,E1 -16539.316,E2 -16539.316} C_VEL
LIN {X 0,Y 298.53,Z 681.09,A -85,B 0,C 180,E1 -16542.179,E2 -16542.179} C_VEL
LIN {X 0,Y 298.585,Z 681.102,A -85,B 0,C 180,E1 -16544.995,E2 -16544.995} C_VEL
LIN {X 0,Y 298.585,Z 681.1,A -85,B 0,C 180,E1 -16549.147,E2 -16549.147} C_VEL
LIN {X 0,Y 298.743,Z 681.061,A -85,B 0,C 180,E1 -16551.886,E2 -16551.886} C_VEL
LIN {X 0,Y 298.654,Z 681.095,A -85,B 0,C 180,E1 -16554.599,E2 -16554.599} C_VEL
LIN {X 0,Y 298.917,Z 681.047,A -85,B 0,C 180,E1 -16558.653,E2 -16558.653} C_VEL
LIN {X 0,Y 298.917,Z 681.052,A -85,B 0,C 180,E1 -16561.348,E2 -16561.348} C_VEL
LIN {X 0,Y 298.787,Z 681.061,A -85,B 0,C 180,E1 -16566.754,E2 -16566.754} C_VEL
LIN {X 0,Y 298.743,Z 681.058,A -85,B 0,C 180,E1 -16567.904,E2 -16567.904} C_VEL
LIN {X 0,Y 298.064,Z 681.15,A -85,B 0,C 180,E1 -16569.028,E2 -16569.028} C_VEL
LIN {X 0,Y 295.104,Z 681.534,A -85,B 0,C 180,E1 -16570.854,E2 -16570.854} C_VEL
LIN {X 0,Y 292.611,Z 681.832,A -85,B 0,C 180,E1 -16572.336,E2 -16572.336} C_VEL
LIN {X 0,Y 291.576,Z 681.955,A -85,B 0,C 180,E1 -16573.487,E2 -16573.487} C_VEL
LIN {X 0,Y 291.511,Z 681.966,A -85,B 0,C 180,E1 -16573.877,E2 -16573.877} C_VEL
LIN {X 0,Y 291.48,Z 681.973,A -85,B 0,C 180,E1 -16576.819,E2 -16576.819} C_VEL
LIN {X 0,Y 291.445,Z 681.993,A -85,B 0,C 180,E1 -16579.876,E2 -16579.876} C_VEL
LIN {X 0,Y 291.394,Z 681.997,A -85,B 0,C 180,E1 -16584.206,E2 -16584.206} C_VEL
LIN {X 0,Y 291.416,Z 681.939,A -85,B 0,C 180,E1 -16587.272,E2 -16587.272} C_VEL
LIN {X 0,Y 291.331,Z 681.952,A -85,B 0,C 180,E1 -16590.438,E2 -16590.438} C_VEL
LIN {X 0,Y 291.339,Z 681.985,A -85,B 0,C 180,E1 -16593.699,E2 -16593.699} C_VEL
LIN {X 0,Y 291.403,Z 682.091,A -85,B 0,C 180,E1 -16596.113,E2 -16596.113} C_VEL
LIN {X 0,Y 292.625,Z 685.792,A -85,B 0,C 180,E1 -16597.902,E2 -16597.902} C_VEL
LIN {X 0,Y 295.504,Z 690.489,A -85,B 0,C 180,E1 -16598.876,E2 -16598.876} C_VEL
LIN {X 0,Y 297.309,Z 693.051,A -85,B 0,C 180,E1 -16599.398,E2 -16599.398} C_VEL
LIN {X 0,Y 301.497,Z 699.462,A -85,B 0,C 180,E1 -16600.58,E2 -16600.58} C_VEL
LIN {X 0,Y 305.21,Z 705.319,A -85,B 0,C 180,E1 -16601.584,E2 -16601.584} C_VEL
LIN {X 0,Y 308.158,Z 710.135,A -85,B 0,C 180,E1 -16602.357,E2 -16602.357} C_VEL
LIN {X 0,Y 315.533,Z 722.891,A -85,B 0,C 180,E1 -16604.203,E2 -16604.203} C_VEL
LIN {X 0,Y 322.942,Z 737.043,A -85,B 0,C 180,E1 -16605.959,E2 -16605.959} C_VEL
LIN {X 0,Y 330.372,Z 752.846,A -85,B 0,C 180,E1 -16607.639,E2 -16607.639} C_VEL
LIN {X 0,Y 332.327,Z 757.318,A -85,B 0,C 180,E1 -16608.071,E2 -16608.071} C_VEL
LIN {X 0,Y 326.361,Z 890.931,A -85,B 0,C 180,E1 -16610.976,E2 -16610.976} C_VEL
LIN {X 0,Y 325.346,Z 903.573,A -85,B 0,C 180,E1 -16611.361,E2 -16611.361} C_VEL
LIN {X 0,Y 323.77,Z 916.673,A -85,B 0,C 180,E1 -16611.883,E2 -16611.883} C_VEL
LIN {X 0,Y 321.968,Z 929.041,A -85,B 0,C 180,E1 -16612.523,E2 -16612.523} C_VEL
LIN {X 0,Y 320.143,Z 940.428,A -85,B 0,C 180,E1 -16613.259,E2 -16613.259} C_VEL
LIN {X 0,Y 317.541,Z 953.659,A -85,B 0,C 180,E1 -16614.287,E2 -16614.287} C_VEL
LIN {X 0,Y 314.808,Z 966.396,A -85,B 0,C 180,E1 -16615.495,E2 -16615.495} C_VEL
LIN {X 0,Y 312.047,Z 978.047,A -85,B 0,C 180,E1 -16616.805,E2 -16616.805} C_VEL
LIN {X 0,Y 309.038,Z 989.274,A -85,B 0,C 180,E1 -16618.272,E2 -16618.272} C_VEL
LIN {X 0,Y 306.517,Z 998.685,A -85,B 0,C 180,E1 -16619.707,E2 -16619.707} C_VEL
LIN {X 0,Y 303.658,Z 1008.784,A -85,B 0,C 180,E1 -16621.487,E2 -16621.487} C_VEL
LIN {X 0,Y 301.085,Z 1017.688,A -85,B 0,C 180,E1 -16623.3,E2 -16623.3} C_VEL
LIN {X 0,Y 298.574,Z 1026.212,A -85,B 0,C 180,E1 -16625.304,E2 -16625.304} C_VEL
LIN {X 0,Y 296.093,Z 1034.814,A -85,B 0,C 180,E1 -16627.681,E2 -16627.681} C_VEL
LIN {X 0,Y 294.344,Z 1041.247,A -85,B 0,C 180,E1 -16629.745,E2 -16629.745} C_VEL
LIN {X 0,Y 292.4,Z 1048.51,A -85,B 0,C 180,E1 -16632.516,E2 -16632.516} C_VEL
LIN {X 0,Y 291.234,Z 1053.634,A -85,B 0,C 180,E1 -16634.856,E2 -16634.856} C_VEL
LIN {X 0,Y 290.362,Z 1058.268,A -85,B 0,C 180,E1 -16637.418,E2 -16637.418} C_VEL
LIN {X 0,Y 289.704,Z 1062.269,A -85,B 0,C 180,E1 -16640.223,E2 -16640.223} C_VEL
LIN {X 0,Y 289.476,Z 1065.231,A -85,B 0,C 180,E1 -16643.028,E2 -16643.028} C_VEL
LIN {X 0,Y 289.408,Z 1066.583,A -85,B 0,C 180,E1 -16644.651,E2 -16644.651} C_VEL
LIN {X 0,Y 289.416,Z 1067.891,A -85,B 0,C 180,E1 -16647.216,E2 -16647.216} C_VEL
LIN {X 0,Y 289.434,Z 1068.379,A -85,B 0,C 180,E1 -16650,E2 -16650} C_VEL
LIN {X 0,Y 289.416,Z 1067.891,A -85,B 0,C 180,E1 -16652.784,E2 -16652.784} C_VEL
LIN {X 0,Y 289.433,Z 1066.42,A -85,B 0,C 180,E1 -16655.574,E2 -16655.574} C_VEL
LIN {X 0,Y 289.552,Z 1063.946,A -85,B 0,C 180,E1 -16658.374,E2 -16658.374} C_VEL
LIN {X 0,Y 290.147,Z 1059.356,A -85,B 0,C 180,E1 -16661.881,E2 -16661.881} C_VEL
LIN {X 0,Y 290.821,Z 1055.865,A -85,B 0,C 180,E1 -16663.984,E2 -16663.984} C_VEL
LIN {X 0,Y 292.007,Z 1050.133,A -85,B 0,C 180,E1 -16666.787,E2 -16666.787} C_VEL
LIN {X 0,Y 293.295,Z 1045.071,A -85,B 0,C 180,E1 -16668.874,E2 -16668.874} C_VEL
LIN {X 0,Y 295.393,Z 1037.303,A -85,B 0,C 180,E1 -16671.552,E2 -16671.552} C_VEL
LIN {X 0,Y 297.422,Z 1030.051,A -85,B 0,C 180,E1 -16673.684,E2 -16673.684} C_VEL
LIN {X 0,Y 299.76,Z 1022.082,A -85,B 0,C 180,E1 -16675.704,E2 -16675.704} C_VEL
LIN {X 0,Y 302.468,Z 1012.971,A -85,B 0,C 180,E1 -16677.691,E2 -16677.691} C_VEL
LIN {X 0,Y 304.897,Z 1004.402,A -85,B 0,C 180,E1 -16679.328,E2 -16679.328} C_VEL
LIN {X 0,Y 308.164,Z 992.538,A -85,B 0,C 180,E1 -16681.253,E2 -16681.253} C_VEL
LIN {X 0,Y 310.886,Z 982.375,A -85,B 0,C 180,E1 -16682.664,E2 -16682.664} C_VEL
LIN {X 0,Y 313.785,Z 970.709,A -85,B 0,C 180,E1 -16684.05,E2 -16684.05} C_VEL
LIN {X 0,Y 316.49,Z 958.685,A -85,B 0,C 180,E1 -16685.264,E2 -16685.264} C_VEL
LIN {X 0,Y 319.018,Z 946.37,A -85,B 0,C 180,E1 -16686.302,E2 -16686.302} C_VEL
LIN {X 0,Y 321.216,Z 933.827,A -85,B 0,C 180,E1 -16687.186,E2 -16687.186} C_VEL
LIN {X 0,Y 323.227,Z 920.401,A -85,B 0,C 180,E1 -16687.945,E2 -16687.945} C_VEL
LIN {X 0,Y 324.904,Z 907.488,A -85,B 0,C 180,E1 -16688.503,E2 -16688.503} C_VEL
LIN {X 0,Y 326.219,Z 894.031,A -85,B 0,C 180,E1 -16688.934,E2 -16688.934} C_VEL
LIN {X 0,Y 327.487,Z 866.329,A -85,B 0,C 180,E1 -16689.589,E2 -16689.589} C_VEL
LIN {X 0,Y 332.322,Z 757.38,A -85,B 0,C 180,E1 -16691.928,E2 -16691.928} C_VEL
LIN {X 0,Y 326.661,Z 744.757,A -85,B 0,C 180,E1 -16693.19,E2 -16693.19} C_VEL
LIN {X 0,Y 318.975,Z 729.263,A -85,B 0,C 180,E1 -16694.971,E2 -16694.971} C_VEL
LIN {X 0,Y 311.392,Z 715.639,A -85,B 0,C 180,E1 -16696.818,E2 -16696.818} C_VEL
LIN {X 0,Y 305.663,Z 705.998,A -85,B 0,C 180,E1 -16698.297,E2 -16698.297} C_VEL
LIN {X 0,Y 301.968,Z 700.211,A -85,B 0,C 180,E1 -16699.29,E2 -16699.29} C_VEL
LIN {X 0,Y 299.254,Z 696.017,A -85,B 0,C 180,E1 -16700.046,E2 -16700.046} C_VEL
LIN {X 0,Y 295.828,Z 690.857,A -85,B 0,C 180,E1 -16701.033,E2 -16701.033} C_VEL
LIN {X 0,Y 292.738,Z 686.113,A -85,B 0,C 180,E1 -16702.01,E2 -16702.01} C_VEL
LIN {X 0,Y 291.897,Z 683.782,A -85,B 0,C 180,E1 -16702.992,E2 -16702.992} C_VEL
LIN {X 0,Y 291.4,Z 682.005,A -85,B 0,C 180,E1 -16703.993,E2 -16703.993} C_VEL
LIN {X 0,Y 291.367,Z 681.991,A -85,B 0,C 180,E1 -16707.95,E2 -16707.95} C_VEL
LIN {X 0,Y 291.376,Z 681.931,A -85,B 0,C 180,E1 -16711.157,E2 -16711.157} C_VEL
LIN {X 0,Y 291.409,Z 681.978,A -85,B 0,C 180,E1 -16714.271,E2 -16714.271} C_VEL
LIN {X 0,Y 291.376,Z 681.983,A -85,B 0,C 180,E1 -16717.299,E2 -16717.299} C_VEL
LIN {X 0,Y 291.456,Z 681.99,A -85,B 0,C 180,E1 -16720.27,E2 -16720.27} C_VEL
LIN {X 0,Y 291.534,Z 681.985,A -85,B 0,C 180,E1 -16724.634,E2 -16724.634} C_VEL
LIN {X 0,Y 291.531,Z 681.977,A -85,B 0,C 180,E1 -16728.88,E2 -16728.88} C_VEL
LIN {X 0,Y 291.699,Z 681.937,A -85,B 0,C 180,E1 -16731.688,E2 -16731.688} C_VEL
LIN {X 0,Y 291.624,Z 681.968,A -85,B 0,C 180,E1 -16734.468,E2 -16734.468} C_VEL
LIN {X 0,Y 291.883,Z 681.925,A -85,B 0,C 180,E1 -16738.62,E2 -16738.62} C_VEL
